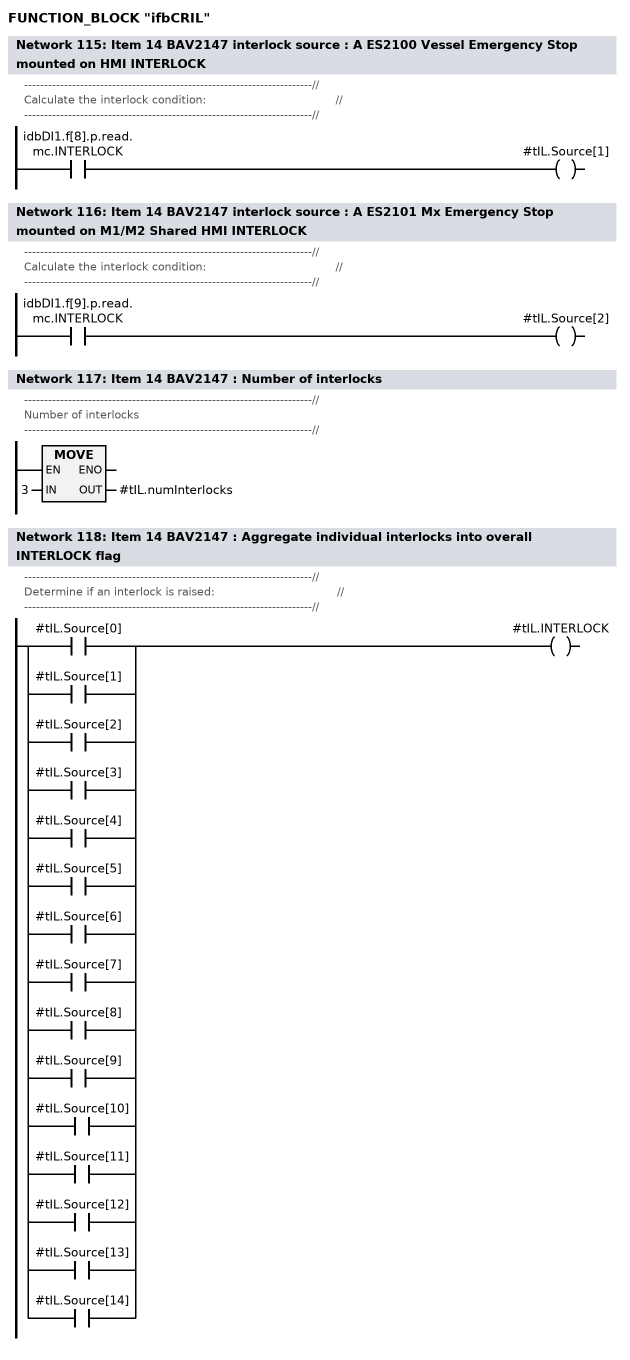
    A idbDI1.f[8].p.read.mc.INTERLOCK;
    = #tIL.Source[1];

NETWORK
TITLE = Item 14 BAV2147 interlock source : A ES2101 Mx Emergency Stop mounted on M1/M2 Shared HMI INTERLOCK
    //------------------------------------------------------------------------//
    // Calculate the interlock condition:                                     //
    //------------------------------------------------------------------------//
    A idbDI1.f[9].p.read.mc.INTERLOCK;
    = #tIL.Source[2];


NETWORK
TITLE = Item 14 BAV2147 : Number of interlocks
    //------------------------------------------------------------------------//
    // Number of interlocks
    //------------------------------------------------------------------------//
    L 3;
    T #tIL.numInterlocks;

NETWORK
TITLE = Item 14 BAV2147 : Aggregate individual interlocks into overall INTERLOCK flag
    //------------------------------------------------------------------------//
    // Determine if an interlock is raised:                                   //
    //------------------------------------------------------------------------//
    O #tIL.Source[0];
    O #tIL.Source[1];
    O #tIL.Source[2];
    O #tIL.Source[3];
    O #tIL.Source[4];
    O #tIL.Source[5];
    O #tIL.Source[6];
    O #tIL.Source[7];
    O #tIL.Source[8];
    O #tIL.Source[9];
    O #tIL.Source[10];
    O #tIL.Source[11];
    O #tIL.Source[12];
    O #tIL.Source[13];
    O #tIL.Source[14];
    = #tIL.INTERLOCK;

NETWORK
TITLE = Item 14 BAV2147 : Update the instance data
    //------------------------------------------------------------------------//
    // Update the instance DB with the calculated interlock flags:            //
    //------------------------------------------------------------------------//
    CALL MOVE
    {value_type := 'Variant'}
    (   IN                   := #tIL ,
        OUT                  := #p[14]
    );

NETWORK
TITLE = Item 15 BAV2149 : SMFLx CIP Drain Valve initialise variables
    //------------------------------------------------------------------------//
    // CRITICAL INTERLOCK   CRITICAL INTERLOCK   CRITICAL INTERLOCK   CRITICA //
    // CRITICAL INTERLOCK   CRITICAL INTERLOCK   CRITICAL INTERLOCK   CRITICA //
    //                                                                        //
    // Clear the interlock flag:                                              //
    //------------------------------------------------------------------------//
    A "alwaysLow";
    = #tIL.INTERLOCK;

    //------------------------------------------------------------------------//
    // Clear all interlock values to initialise them to off:                  //
    //------------------------------------------------------------------------//
    CALL FILL_BLK
    {value_type := 'Bool', count_type := 'UInt'}
    (   IN                   := 0 ,
        COUNT                := 15 ,
        OUT                  := #tIL.Source[0]
    );


NETWORK
TITLE = Item 15 BAV2149 interlock source : A RD2101 Vessel Burst Disc ALARM
    //------------------------------------------------------------------------//
    // Calculate the interlock condition:                                     //
    //------------------------------------------------------------------------//
    A idbDI1.f[14].p.read.mc.INTERLOCK;
    = #tIL.Source[0];

NETWORK
TITLE = Item 15 BAV2149 interlock source : A ES2100 Vessel Emergency Stop mounted on HMI INTERLOCK
    //------------------------------------------------------------------------//
    // Calculate the interlock condition:                                     //
    //------------------------------------------------------------------------//
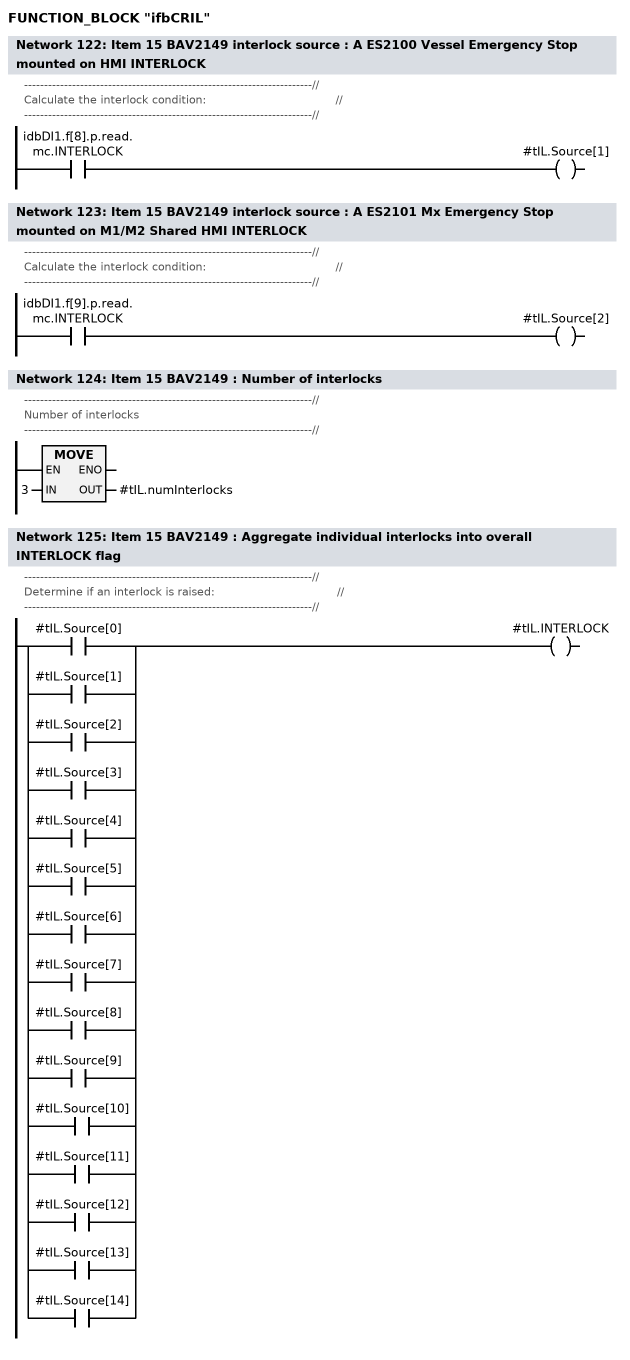
    A idbDI1.f[8].p.read.mc.INTERLOCK;
    = #tIL.Source[1];

NETWORK
TITLE = Item 15 BAV2149 interlock source : A ES2101 Mx Emergency Stop mounted on M1/M2 Shared HMI INTERLOCK
    //------------------------------------------------------------------------//
    // Calculate the interlock condition:                                     //
    //------------------------------------------------------------------------//
    A idbDI1.f[9].p.read.mc.INTERLOCK;
    = #tIL.Source[2];


NETWORK
TITLE = Item 15 BAV2149 : Number of interlocks
    //------------------------------------------------------------------------//
    // Number of interlocks
    //------------------------------------------------------------------------//
    L 3;
    T #tIL.numInterlocks;

NETWORK
TITLE = Item 15 BAV2149 : Aggregate individual interlocks into overall INTERLOCK flag
    //------------------------------------------------------------------------//
    // Determine if an interlock is raised:                                   //
    //------------------------------------------------------------------------//
    O #tIL.Source[0];
    O #tIL.Source[1];
    O #tIL.Source[2];
    O #tIL.Source[3];
    O #tIL.Source[4];
    O #tIL.Source[5];
    O #tIL.Source[6];
    O #tIL.Source[7];
    O #tIL.Source[8];
    O #tIL.Source[9];
    O #tIL.Source[10];
    O #tIL.Source[11];
    O #tIL.Source[12];
    O #tIL.Source[13];
    O #tIL.Source[14];
    = #tIL.INTERLOCK;

NETWORK
TITLE = Item 15 BAV2149 : Update the instance data
    //------------------------------------------------------------------------//
    // Update the instance DB with the calculated interlock flags:            //
    //------------------------------------------------------------------------//
    CALL MOVE
    {value_type := 'Variant'}
    (   IN                   := #tIL ,
        OUT                  := #p[15]
    );

NETWORK
TITLE = Item 16 BAV2167 : MMFLx Cooling Water Supply Drain Valve initialise variables
    //------------------------------------------------------------------------//
    // CRITICAL INTERLOCK   CRITICAL INTERLOCK   CRITICAL INTERLOCK   CRITICA //
    // CRITICAL INTERLOCK   CRITICAL INTERLOCK   CRITICAL INTERLOCK   CRITICA //
    //                                                                        //
    // Clear the interlock flag:                                              //
    //------------------------------------------------------------------------//
    A "alwaysLow";
    = #tIL.INTERLOCK;

    //------------------------------------------------------------------------//
    // Clear all interlock values to initialise them to off:                  //
    //------------------------------------------------------------------------//
    CALL FILL_BLK
    {value_type := 'Bool', count_type := 'UInt'}
    (   IN                   := 0 ,
        COUNT                := 15 ,
        OUT                  := #tIL.Source[0]
    );


NETWORK
TITLE = Item 16 BAV2167 interlock source : A RD2101 Vessel Burst Disc ALARM
    //------------------------------------------------------------------------//
    // Calculate the interlock condition:                                     //
    //------------------------------------------------------------------------//
    A idbDI1.f[14].p.read.mc.INTERLOCK;
    = #tIL.Source[0];

NETWORK
TITLE = Item 16 BAV2167 interlock source : A ES2100 Vessel Emergency Stop mounted on HMI INTERLOCK
    //------------------------------------------------------------------------//
    // Calculate the interlock condition:                                     //
    //------------------------------------------------------------------------//
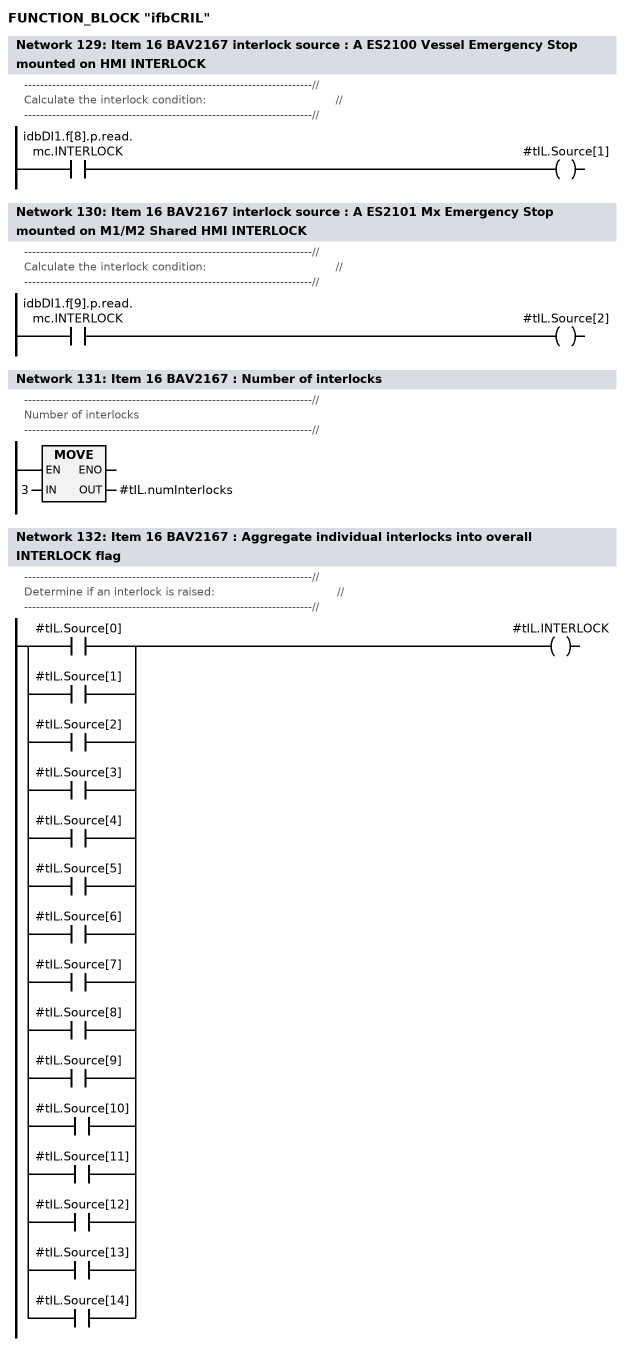
    A idbDI1.f[8].p.read.mc.INTERLOCK;
    = #tIL.Source[1];

NETWORK
TITLE = Item 16 BAV2167 interlock source : A ES2101 Mx Emergency Stop mounted on M1/M2 Shared HMI INTERLOCK
    //------------------------------------------------------------------------//
    // Calculate the interlock condition:                                     //
    //------------------------------------------------------------------------//
    A idbDI1.f[9].p.read.mc.INTERLOCK;
    = #tIL.Source[2];


NETWORK
TITLE = Item 16 BAV2167 : Number of interlocks
    //------------------------------------------------------------------------//
    // Number of interlocks
    //------------------------------------------------------------------------//
    L 3;
    T #tIL.numInterlocks;

NETWORK
TITLE = Item 16 BAV2167 : Aggregate individual interlocks into overall INTERLOCK flag
    //------------------------------------------------------------------------//
    // Determine if an interlock is raised:                                   //
    //------------------------------------------------------------------------//
    O #tIL.Source[0];
    O #tIL.Source[1];
    O #tIL.Source[2];
    O #tIL.Source[3];
    O #tIL.Source[4];
    O #tIL.Source[5];
    O #tIL.Source[6];
    O #tIL.Source[7];
    O #tIL.Source[8];
    O #tIL.Source[9];
    O #tIL.Source[10];
    O #tIL.Source[11];
    O #tIL.Source[12];
    O #tIL.Source[13];
    O #tIL.Source[14];
    = #tIL.INTERLOCK;

NETWORK
TITLE = Item 16 BAV2167 : Update the instance data
    //------------------------------------------------------------------------//
    // Update the instance DB with the calculated interlock flags:            //
    //------------------------------------------------------------------------//
    CALL MOVE
    {value_type := 'Variant'}
    (   IN                   := #tIL ,
        OUT                  := #p[16]
    );

NETWORK
TITLE = Item 17 BAV2169 : MMFLx Cooling Water Return Drain Valve initialise variables
    //------------------------------------------------------------------------//
    // CRITICAL INTERLOCK   CRITICAL INTERLOCK   CRITICAL INTERLOCK   CRITICA //
    // CRITICAL INTERLOCK   CRITICAL INTERLOCK   CRITICAL INTERLOCK   CRITICA //
    //                                                                        //
    // Clear the interlock flag:                                              //
    //------------------------------------------------------------------------//
    A "alwaysLow";
    = #tIL.INTERLOCK;

    //------------------------------------------------------------------------//
    // Clear all interlock values to initialise them to off:                  //
    //------------------------------------------------------------------------//
    CALL FILL_BLK
    {value_type := 'Bool', count_type := 'UInt'}
    (   IN                   := 0 ,
        COUNT                := 15 ,
        OUT                  := #tIL.Source[0]
    );


NETWORK
TITLE = Item 17 BAV2169 interlock source : A RD2101 Vessel Burst Disc ALARM
    //------------------------------------------------------------------------//
    // Calculate the interlock condition:                                     //
    //------------------------------------------------------------------------//
    A idbDI1.f[14].p.read.mc.INTERLOCK;
    = #tIL.Source[0];

NETWORK
TITLE = Item 17 BAV2169 interlock source : A ES2100 Vessel Emergency Stop mounted on HMI INTERLOCK
    //------------------------------------------------------------------------//
    // Calculate the interlock condition:                                     //
    //------------------------------------------------------------------------//
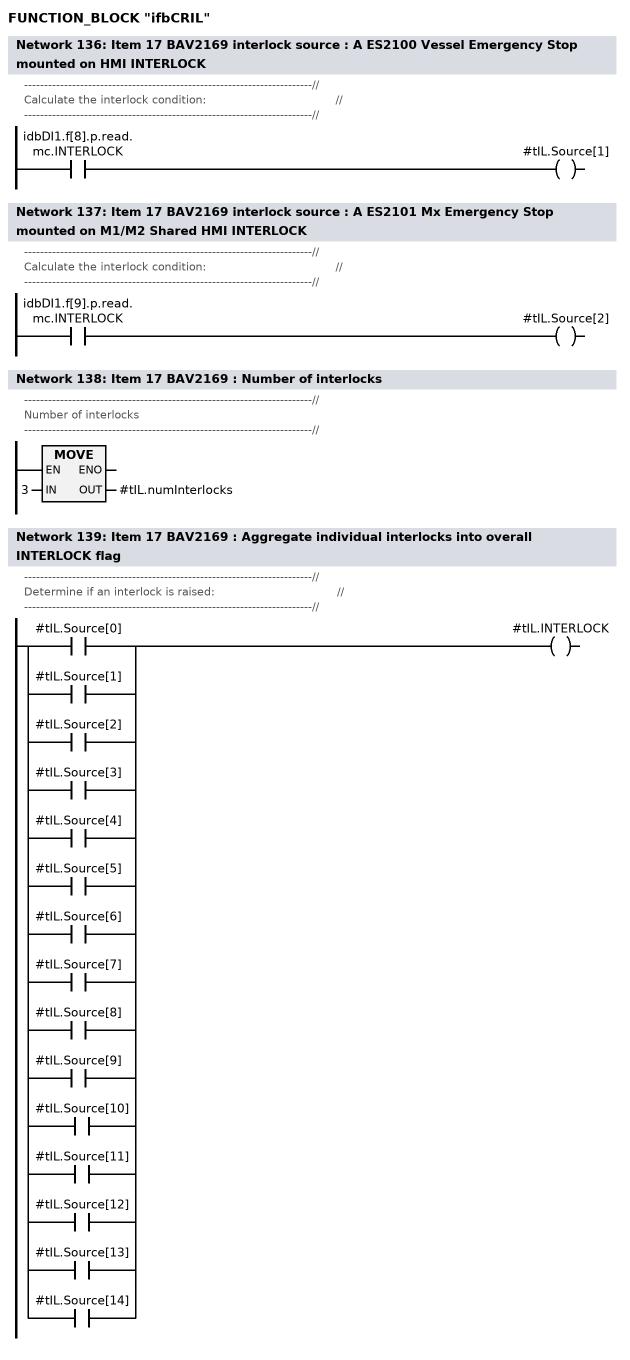
    A idbDI1.f[8].p.read.mc.INTERLOCK;
    = #tIL.Source[1];

NETWORK
TITLE = Item 17 BAV2169 interlock source : A ES2101 Mx Emergency Stop mounted on M1/M2 Shared HMI INTERLOCK
    //------------------------------------------------------------------------//
    // Calculate the interlock condition:                                     //
    //------------------------------------------------------------------------//
    A idbDI1.f[9].p.read.mc.INTERLOCK;
    = #tIL.Source[2];


NETWORK
TITLE = Item 17 BAV2169 : Number of interlocks
    //------------------------------------------------------------------------//
    // Number of interlocks
    //------------------------------------------------------------------------//
    L 3;
    T #tIL.numInterlocks;

NETWORK
TITLE = Item 17 BAV2169 : Aggregate individual interlocks into overall INTERLOCK flag
    //------------------------------------------------------------------------//
    // Determine if an interlock is raised:                                   //
    //------------------------------------------------------------------------//
    O #tIL.Source[0];
    O #tIL.Source[1];
    O #tIL.Source[2];
    O #tIL.Source[3];
    O #tIL.Source[4];
    O #tIL.Source[5];
    O #tIL.Source[6];
    O #tIL.Source[7];
    O #tIL.Source[8];
    O #tIL.Source[9];
    O #tIL.Source[10];
    O #tIL.Source[11];
    O #tIL.Source[12];
    O #tIL.Source[13];
    O #tIL.Source[14];
    = #tIL.INTERLOCK;

NETWORK
TITLE = Item 17 BAV2169 : Update the instance data
    //------------------------------------------------------------------------//
    // Update the instance DB with the calculated interlock flags:            //
    //------------------------------------------------------------------------//
    CALL MOVE
    {value_type := 'Variant'}
    (   IN                   := #tIL ,
        OUT                  := #p[17]
    );

NETWORK
TITLE = Item 18 BAV3139 : Vent line drain valve initialise variables
    //------------------------------------------------------------------------//
    // CRITICAL INTERLOCK   CRITICAL INTERLOCK   CRITICAL INTERLOCK   CRITICA //
    // CRITICAL INTERLOCK   CRITICAL INTERLOCK   CRITICAL INTERLOCK   CRITICA //
    //                                                                        //
    // Clear the interlock flag:                                              //
    //------------------------------------------------------------------------//
    A "alwaysLow";
    = #tIL.INTERLOCK;

    //------------------------------------------------------------------------//
    // Clear all interlock values to initialise them to off:                  //
    //------------------------------------------------------------------------//
    CALL FILL_BLK
    {value_type := 'Bool', count_type := 'UInt'}
    (   IN                   := 0 ,
        COUNT                := 15 ,
        OUT                  := #tIL.Source[0]
    );


NETWORK
TITLE = Item 18 BAV3139 interlock source : A RD3101 Vessel Burst Disc ALARM
    //------------------------------------------------------------------------//
    // Calculate the interlock condition:                                     //
    //------------------------------------------------------------------------//
    A idbDI1.f[15].p.read.mc.INTERLOCK;
    = #tIL.Source[0];

NETWORK
TITLE = Item 18 BAV3139 interlock source : A ES3100 Vessel Emergency Stop mounted on HMI INTERLOCK
    //------------------------------------------------------------------------//
    // Calculate the interlock condition:                                     //
    //------------------------------------------------------------------------//
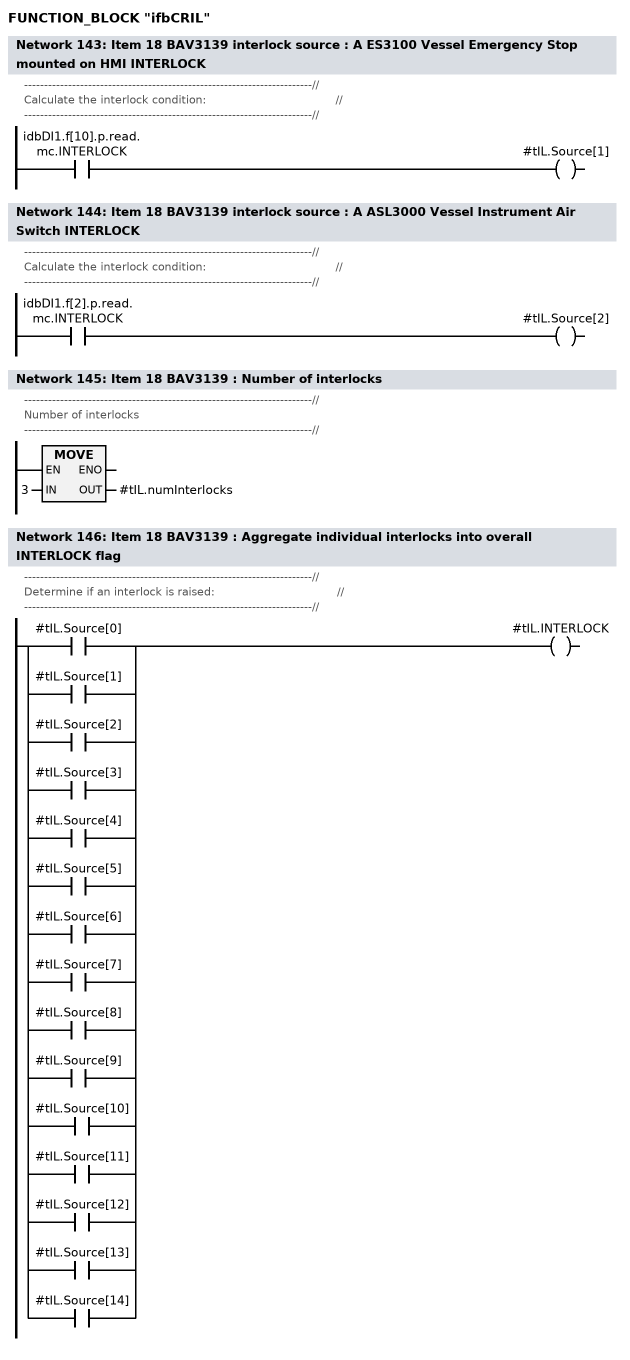
    A idbDI1.f[10].p.read.mc.INTERLOCK;
    = #tIL.Source[1];

NETWORK
TITLE = Item 18 BAV3139 interlock source : A ASL3000 Vessel Instrument Air Switch INTERLOCK
    //------------------------------------------------------------------------//
    // Calculate the interlock condition:                                     //
    //------------------------------------------------------------------------//
    A idbDI1.f[2].p.read.mc.INTERLOCK;
    = #tIL.Source[2];


NETWORK
TITLE = Item 18 BAV3139 : Number of interlocks
    //------------------------------------------------------------------------//
    // Number of interlocks
    //------------------------------------------------------------------------//
    L 3;
    T #tIL.numInterlocks;

NETWORK
TITLE = Item 18 BAV3139 : Aggregate individual interlocks into overall INTERLOCK flag
    //------------------------------------------------------------------------//
    // Determine if an interlock is raised:                                   //
    //------------------------------------------------------------------------//
    O #tIL.Source[0];
    O #tIL.Source[1];
    O #tIL.Source[2];
    O #tIL.Source[3];
    O #tIL.Source[4];
    O #tIL.Source[5];
    O #tIL.Source[6];
    O #tIL.Source[7];
    O #tIL.Source[8];
    O #tIL.Source[9];
    O #tIL.Source[10];
    O #tIL.Source[11];
    O #tIL.Source[12];
    O #tIL.Source[13];
    O #tIL.Source[14];
    = #tIL.INTERLOCK;

NETWORK
TITLE = Item 18 BAV3139 : Update the instance data
    //------------------------------------------------------------------------//
    // Update the instance DB with the calculated interlock flags:            //
    //------------------------------------------------------------------------//
    CALL MOVE
    {value_type := 'Variant'}
    (   IN                   := #tIL ,
        OUT                  := #p[18]
    );

NETWORK
TITLE = Item 19 BAV3141 : Vent Filter Drain valve initialise variables
    //------------------------------------------------------------------------//
    // CRITICAL INTERLOCK   CRITICAL INTERLOCK   CRITICAL INTERLOCK   CRITICA //
    // CRITICAL INTERLOCK   CRITICAL INTERLOCK   CRITICAL INTERLOCK   CRITICA //
    //                                                                        //
    // Clear the interlock flag:                                              //
    //------------------------------------------------------------------------//
    A "alwaysLow";
    = #tIL.INTERLOCK;

    //------------------------------------------------------------------------//
    // Clear all interlock values to initialise them to off:                  //
    //------------------------------------------------------------------------//
    CALL FILL_BLK
    {value_type := 'Bool', count_type := 'UInt'}
    (   IN                   := 0 ,
        COUNT                := 15 ,
        OUT                  := #tIL.Source[0]
    );


NETWORK
TITLE = Item 19 BAV3141 interlock source : A RD3101 Vessel Burst Disc ALARM
    //------------------------------------------------------------------------//
    // Calculate the interlock condition:                                     //
    //------------------------------------------------------------------------//
    A idbDI1.f[15].p.read.mc.INTERLOCK;
    = #tIL.Source[0];

NETWORK
TITLE = Item 19 BAV3141 interlock source : A ES3100 Vessel Emergency Stop mounted on HMI INTERLOCK
    //------------------------------------------------------------------------//
    // Calculate the interlock condition:                                     //
    //------------------------------------------------------------------------//
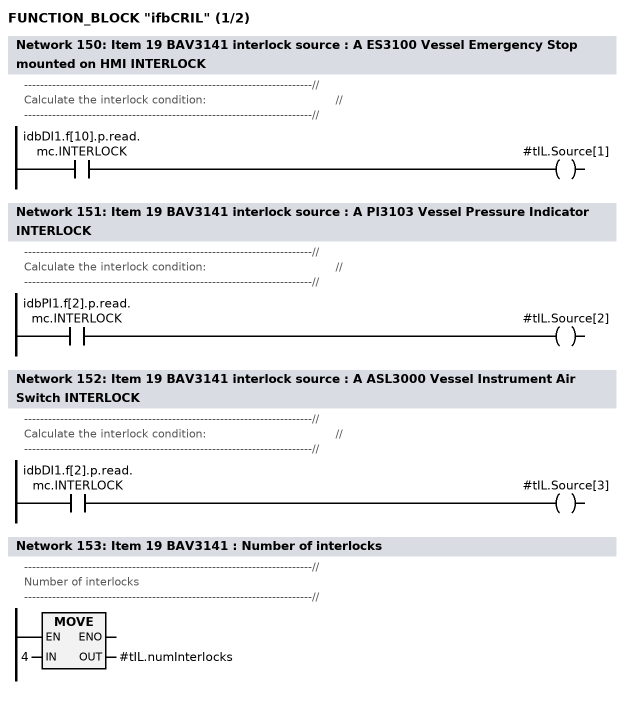
    A idbDI1.f[10].p.read.mc.INTERLOCK;
    = #tIL.Source[1];

NETWORK
TITLE = Item 19 BAV3141 interlock source : A PI3103 Vessel Pressure Indicator INTERLOCK
    //------------------------------------------------------------------------//
    // Calculate the interlock condition:                                     //
    //------------------------------------------------------------------------//
    A idbPI1.f[2].p.read.mc.INTERLOCK;
    = #tIL.Source[2];

NETWORK
TITLE = Item 19 BAV3141 interlock source : A ASL3000 Vessel Instrument Air Switch INTERLOCK
    //------------------------------------------------------------------------//
    // Calculate the interlock condition:                                     //
    //------------------------------------------------------------------------//
    A idbDI1.f[2].p.read.mc.INTERLOCK;
    = #tIL.Source[3];


NETWORK
TITLE = Item 19 BAV3141 : Number of interlocks
    //------------------------------------------------------------------------//
    // Number of interlocks
    //------------------------------------------------------------------------//
    L 4;
    T #tIL.numInterlocks;

NETWORK
TITLE = Item 19 BAV3141 : Aggregate individual interlocks into overall INTERLOCK flag
    //------------------------------------------------------------------------//
    // Determine if an interlock is raised:                                   //
    //------------------------------------------------------------------------//
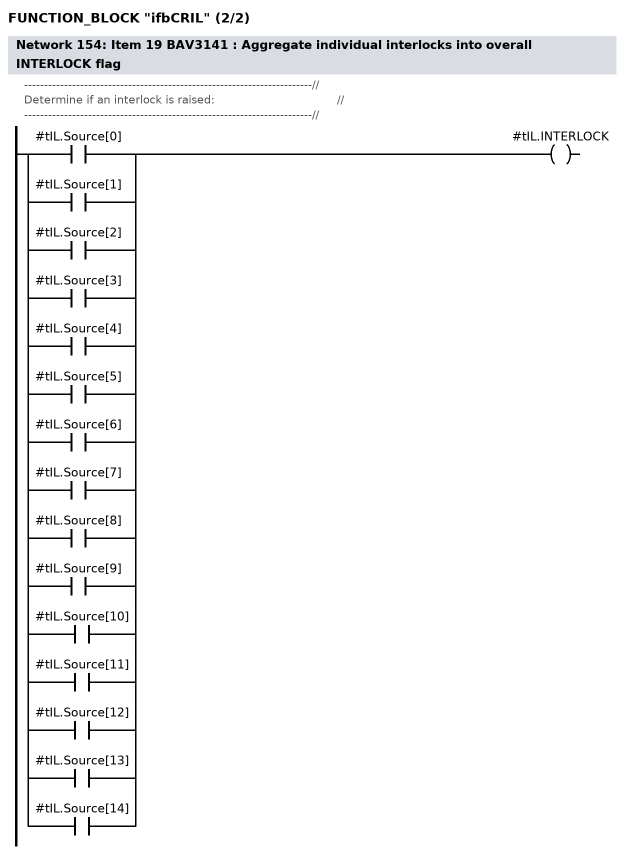
    O #tIL.Source[0];
    O #tIL.Source[1];
    O #tIL.Source[2];
    O #tIL.Source[3];
    O #tIL.Source[4];
    O #tIL.Source[5];
    O #tIL.Source[6];
    O #tIL.Source[7];
    O #tIL.Source[8];
    O #tIL.Source[9];
    O #tIL.Source[10];
    O #tIL.Source[11];
    O #tIL.Source[12];
    O #tIL.Source[13];
    O #tIL.Source[14];
    = #tIL.INTERLOCK;

NETWORK
TITLE = Item 19 BAV3141 : Update the instance data
    //------------------------------------------------------------------------//
    // Update the instance DB with the calculated interlock flags:            //
    //------------------------------------------------------------------------//
    CALL MOVE
    {value_type := 'Variant'}
    (   IN                   := #tIL ,
        OUT                  := #p[19]
    );

NETWORK
TITLE = Item 20 BAV3143 : SIP Condensate Drain Valve initialise variables
    //------------------------------------------------------------------------//
    // CRITICAL INTERLOCK   CRITICAL INTERLOCK   CRITICAL INTERLOCK   CRITICA //
    // CRITICAL INTERLOCK   CRITICAL INTERLOCK   CRITICAL INTERLOCK   CRITICA //
    //                                                                        //
    // Clear the interlock flag:                                              //
    //------------------------------------------------------------------------//
    A "alwaysLow";
    = #tIL.INTERLOCK;

    //------------------------------------------------------------------------//
    // Clear all interlock values to initialise them to off:                  //
    //------------------------------------------------------------------------//
    CALL FILL_BLK
    {value_type := 'Bool', count_type := 'UInt'}
    (   IN                   := 0 ,
        COUNT                := 15 ,
        OUT                  := #tIL.Source[0]
    );


NETWORK
TITLE = Item 20 BAV3143 interlock source : A RD3101 Vessel Burst Disc ALARM
    //------------------------------------------------------------------------//
    // Calculate the interlock condition:                                     //
    //------------------------------------------------------------------------//
    A idbDI1.f[15].p.read.mc.INTERLOCK;
    = #tIL.Source[0];

NETWORK
TITLE = Item 20 BAV3143 interlock source : A ES3100 Vessel Emergency Stop mounted on HMI INTERLOCK
    //------------------------------------------------------------------------//
    // Calculate the interlock condition:                                     //
    //------------------------------------------------------------------------//
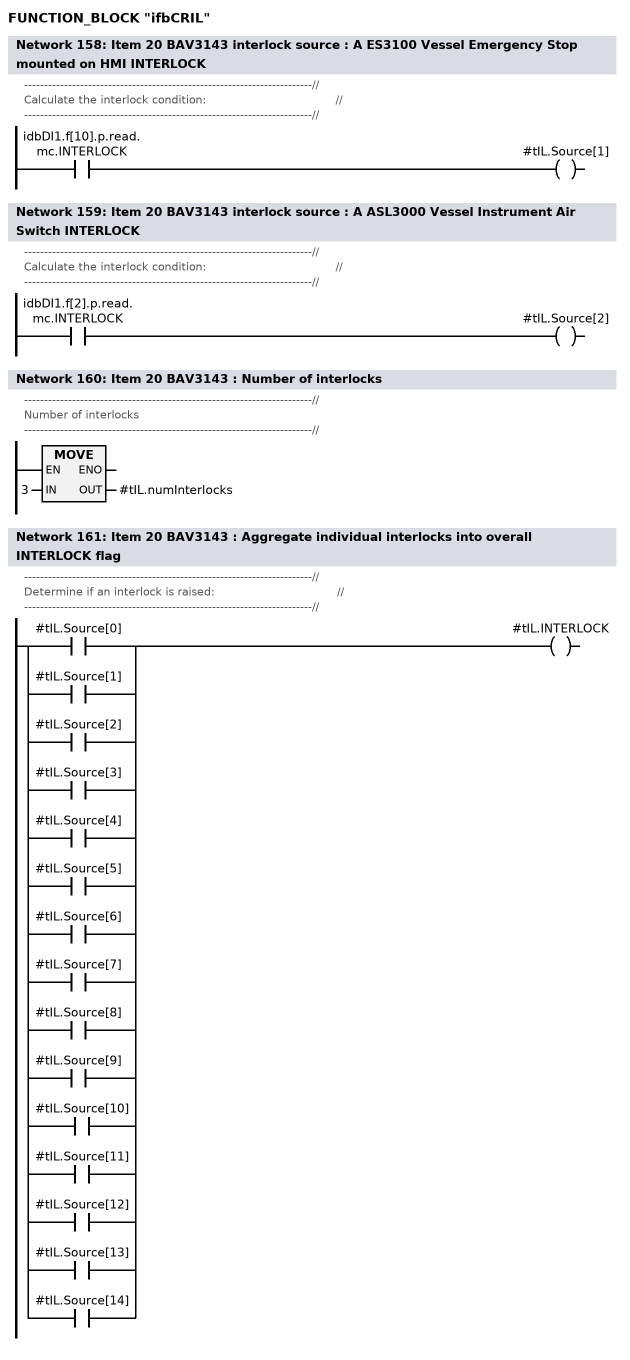
    A idbDI1.f[10].p.read.mc.INTERLOCK;
    = #tIL.Source[1];

NETWORK
TITLE = Item 20 BAV3143 interlock source : A ASL3000 Vessel Instrument Air Switch INTERLOCK
    //------------------------------------------------------------------------//
    // Calculate the interlock condition:                                     //
    //------------------------------------------------------------------------//
    A idbDI1.f[2].p.read.mc.INTERLOCK;
    = #tIL.Source[2];


NETWORK
TITLE = Item 20 BAV3143 : Number of interlocks
    //------------------------------------------------------------------------//
    // Number of interlocks
    //------------------------------------------------------------------------//
    L 3;
    T #tIL.numInterlocks;

NETWORK
TITLE = Item 20 BAV3143 : Aggregate individual interlocks into overall INTERLOCK flag
    //------------------------------------------------------------------------//
    // Determine if an interlock is raised:                                   //
    //------------------------------------------------------------------------//
    O #tIL.Source[0];
    O #tIL.Source[1];
    O #tIL.Source[2];
    O #tIL.Source[3];
    O #tIL.Source[4];
    O #tIL.Source[5];
    O #tIL.Source[6];
    O #tIL.Source[7];
    O #tIL.Source[8];
    O #tIL.Source[9];
    O #tIL.Source[10];
    O #tIL.Source[11];
    O #tIL.Source[12];
    O #tIL.Source[13];
    O #tIL.Source[14];
    = #tIL.INTERLOCK;

NETWORK
TITLE = Item 20 BAV3143 : Update the instance data
    //------------------------------------------------------------------------//
    // Update the instance DB with the calculated interlock flags:            //
    //------------------------------------------------------------------------//
    CALL MOVE
    {value_type := 'Variant'}
    (   IN                   := #tIL ,
        OUT                  := #p[20]
    );

NETWORK
TITLE = Item 21 BAV3145 : CIP Drain Valve initialise variables
    //------------------------------------------------------------------------//
    // CRITICAL INTERLOCK   CRITICAL INTERLOCK   CRITICAL INTERLOCK   CRITICA //
    // CRITICAL INTERLOCK   CRITICAL INTERLOCK   CRITICAL INTERLOCK   CRITICA //
    //                                                                        //
    // Clear the interlock flag:                                              //
    //------------------------------------------------------------------------//
    A "alwaysLow";
    = #tIL.INTERLOCK;

    //------------------------------------------------------------------------//
    // Clear all interlock values to initialise them to off:                  //
    //------------------------------------------------------------------------//
    CALL FILL_BLK
    {value_type := 'Bool', count_type := 'UInt'}
    (   IN                   := 0 ,
        COUNT                := 15 ,
        OUT                  := #tIL.Source[0]
    );


NETWORK
TITLE = Item 21 BAV3145 interlock source : A RD3101 Vessel Burst Disc ALARM
    //------------------------------------------------------------------------//
    // Calculate the interlock condition:                                     //
    //------------------------------------------------------------------------//
    A idbDI1.f[15].p.read.mc.INTERLOCK;
    = #tIL.Source[0];

NETWORK
TITLE = Item 21 BAV3145 interlock source : A ES3100 Vessel Emergency Stop mounted on HMI INTERLOCK
    //------------------------------------------------------------------------//
    // Calculate the interlock condition:                                     //
    //------------------------------------------------------------------------//
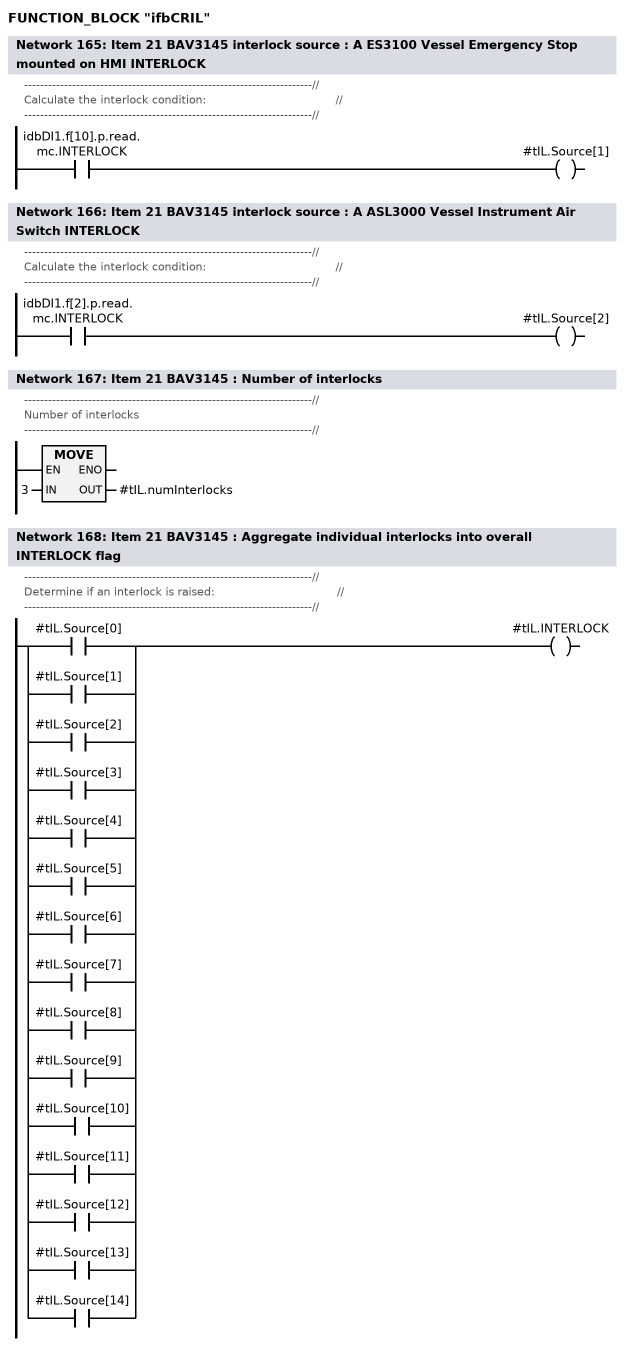
    A idbDI1.f[10].p.read.mc.INTERLOCK;
    = #tIL.Source[1];

NETWORK
TITLE = Item 21 BAV3145 interlock source : A ASL3000 Vessel Instrument Air Switch INTERLOCK
    //------------------------------------------------------------------------//
    // Calculate the interlock condition:                                     //
    //------------------------------------------------------------------------//
    A idbDI1.f[2].p.read.mc.INTERLOCK;
    = #tIL.Source[2];


NETWORK
TITLE = Item 21 BAV3145 : Number of interlocks
    //------------------------------------------------------------------------//
    // Number of interlocks
    //------------------------------------------------------------------------//
    L 3;
    T #tIL.numInterlocks;

NETWORK
TITLE = Item 21 BAV3145 : Aggregate individual interlocks into overall INTERLOCK flag
    //------------------------------------------------------------------------//
    // Determine if an interlock is raised:                                   //
    //------------------------------------------------------------------------//
    O #tIL.Source[0];
    O #tIL.Source[1];
    O #tIL.Source[2];
    O #tIL.Source[3];
    O #tIL.Source[4];
    O #tIL.Source[5];
    O #tIL.Source[6];
    O #tIL.Source[7];
    O #tIL.Source[8];
    O #tIL.Source[9];
    O #tIL.Source[10];
    O #tIL.Source[11];
    O #tIL.Source[12];
    O #tIL.Source[13];
    O #tIL.Source[14];
    = #tIL.INTERLOCK;

NETWORK
TITLE = Item 21 BAV3145 : Update the instance data
    //------------------------------------------------------------------------//
    // Update the instance DB with the calculated interlock flags:            //
    //------------------------------------------------------------------------//
    CALL MOVE
    {value_type := 'Variant'}
    (   IN                   := #tIL ,
        OUT                  := #p[21]
    );

NETWORK
TITLE = Item 22 BAV4139 : Vent line drain valve initialise variables
    //------------------------------------------------------------------------//
    // CRITICAL INTERLOCK   CRITICAL INTERLOCK   CRITICAL INTERLOCK   CRITICA //
    // CRITICAL INTERLOCK   CRITICAL INTERLOCK   CRITICAL INTERLOCK   CRITICA //
    //                                                                        //
    // Clear the interlock flag:                                              //
    //------------------------------------------------------------------------//
    A "alwaysLow";
    = #tIL.INTERLOCK;

    //------------------------------------------------------------------------//
    // Clear all interlock values to initialise them to off:                  //
    //------------------------------------------------------------------------//
    CALL FILL_BLK
    {value_type := 'Bool', count_type := 'UInt'}
    (   IN                   := 0 ,
        COUNT                := 15 ,
        OUT                  := #tIL.Source[0]
    );


NETWORK
TITLE = Item 22 BAV4139 interlock source : A RD4101 Vessel Burst Disc ALARM
    //------------------------------------------------------------------------//
    // Calculate the interlock condition:                                     //
    //------------------------------------------------------------------------//
    A idbDI1.f[16].p.read.mc.INTERLOCK;
    = #tIL.Source[0];

NETWORK
TITLE = Item 22 BAV4139 interlock source : A ES4100 Vessel Emergency Stop mounted on HMI INTERLOCK
    //------------------------------------------------------------------------//
    // Calculate the interlock condition:                                     //
    //------------------------------------------------------------------------//
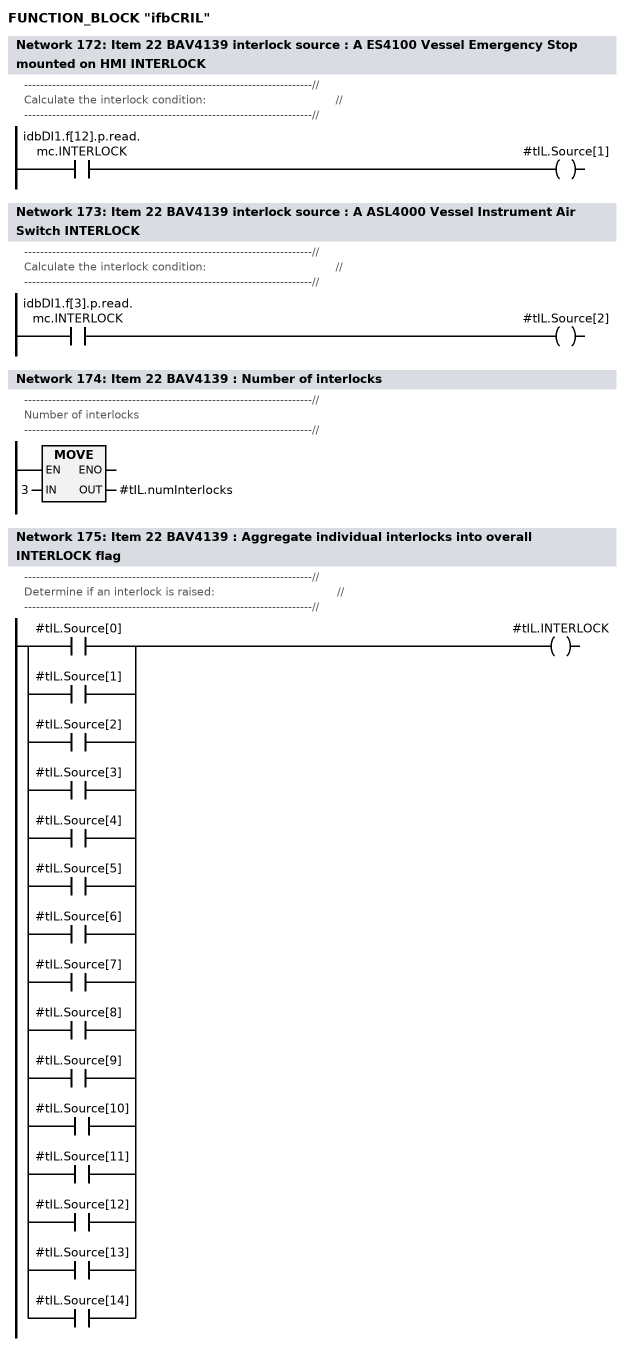
    A idbDI1.f[12].p.read.mc.INTERLOCK;
    = #tIL.Source[1];

NETWORK
TITLE = Item 22 BAV4139 interlock source : A ASL4000 Vessel Instrument Air Switch INTERLOCK
    //------------------------------------------------------------------------//
    // Calculate the interlock condition:                                     //
    //------------------------------------------------------------------------//
    A idbDI1.f[3].p.read.mc.INTERLOCK;
    = #tIL.Source[2];


NETWORK
TITLE = Item 22 BAV4139 : Number of interlocks
    //------------------------------------------------------------------------//
    // Number of interlocks
    //------------------------------------------------------------------------//
    L 3;
    T #tIL.numInterlocks;

NETWORK
TITLE = Item 22 BAV4139 : Aggregate individual interlocks into overall INTERLOCK flag
    //------------------------------------------------------------------------//
    // Determine if an interlock is raised:                                   //
    //------------------------------------------------------------------------//
    O #tIL.Source[0];
    O #tIL.Source[1];
    O #tIL.Source[2];
    O #tIL.Source[3];
    O #tIL.Source[4];
    O #tIL.Source[5];
    O #tIL.Source[6];
    O #tIL.Source[7];
    O #tIL.Source[8];
    O #tIL.Source[9];
    O #tIL.Source[10];
    O #tIL.Source[11];
    O #tIL.Source[12];
    O #tIL.Source[13];
    O #tIL.Source[14];
    = #tIL.INTERLOCK;

NETWORK
TITLE = Item 22 BAV4139 : Update the instance data
    //------------------------------------------------------------------------//
    // Update the instance DB with the calculated interlock flags:            //
    //------------------------------------------------------------------------//
    CALL MOVE
    {value_type := 'Variant'}
    (   IN                   := #tIL ,
        OUT                  := #p[22]
    );

NETWORK
TITLE = Item 23 BAV4141 : Vent Filter Drain valve initialise variables
    //------------------------------------------------------------------------//
    // CRITICAL INTERLOCK   CRITICAL INTERLOCK   CRITICAL INTERLOCK   CRITICA //
    // CRITICAL INTERLOCK   CRITICAL INTERLOCK   CRITICAL INTERLOCK   CRITICA //
    //                                                                        //
    // Clear the interlock flag:                                              //
    //------------------------------------------------------------------------//
    A "alwaysLow";
    = #tIL.INTERLOCK;

    //------------------------------------------------------------------------//
    // Clear all interlock values to initialise them to off:                  //
    //------------------------------------------------------------------------//
    CALL FILL_BLK
    {value_type := 'Bool', count_type := 'UInt'}
    (   IN                   := 0 ,
        COUNT                := 15 ,
        OUT                  := #tIL.Source[0]
    );


NETWORK
TITLE = Item 23 BAV4141 interlock source : A RD4101 Vessel Burst Disc ALARM
    //------------------------------------------------------------------------//
    // Calculate the interlock condition:                                     //
    //------------------------------------------------------------------------//
    A idbDI1.f[16].p.read.mc.INTERLOCK;
    = #tIL.Source[0];

NETWORK
TITLE = Item 23 BAV4141 interlock source : A ES4100 Vessel Emergency Stop mounted on HMI INTERLOCK
    //------------------------------------------------------------------------//
    // Calculate the interlock condition:                                     //
    //------------------------------------------------------------------------//
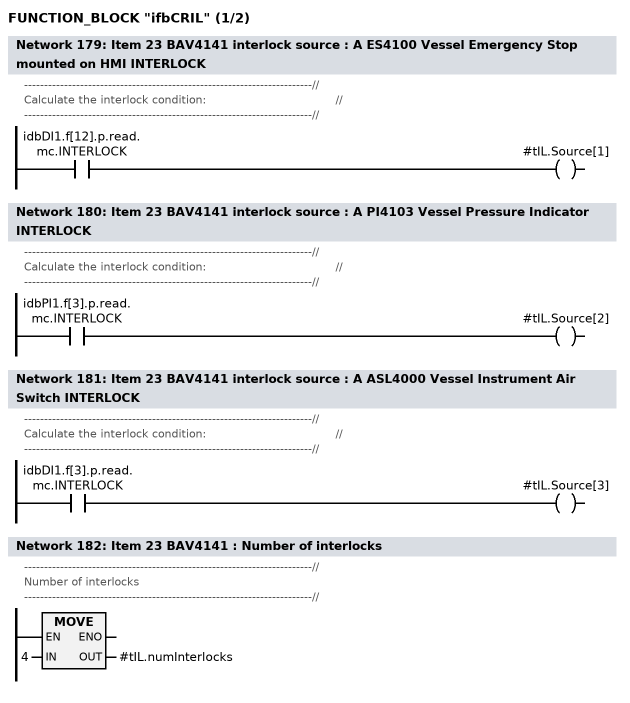
    A idbDI1.f[12].p.read.mc.INTERLOCK;
    = #tIL.Source[1];

NETWORK
TITLE = Item 23 BAV4141 interlock source : A PI4103 Vessel Pressure Indicator INTERLOCK
    //------------------------------------------------------------------------//
    // Calculate the interlock condition:                                     //
    //------------------------------------------------------------------------//
    A idbPI1.f[3].p.read.mc.INTERLOCK;
    = #tIL.Source[2];

NETWORK
TITLE = Item 23 BAV4141 interlock source : A ASL4000 Vessel Instrument Air Switch INTERLOCK
    //------------------------------------------------------------------------//
    // Calculate the interlock condition:                                     //
    //------------------------------------------------------------------------//
    A idbDI1.f[3].p.read.mc.INTERLOCK;
    = #tIL.Source[3];


NETWORK
TITLE = Item 23 BAV4141 : Number of interlocks
    //------------------------------------------------------------------------//
    // Number of interlocks
    //------------------------------------------------------------------------//
    L 4;
    T #tIL.numInterlocks;

NETWORK
TITLE = Item 23 BAV4141 : Aggregate individual interlocks into overall INTERLOCK flag
    //------------------------------------------------------------------------//
    // Determine if an interlock is raised:                                   //
    //------------------------------------------------------------------------//
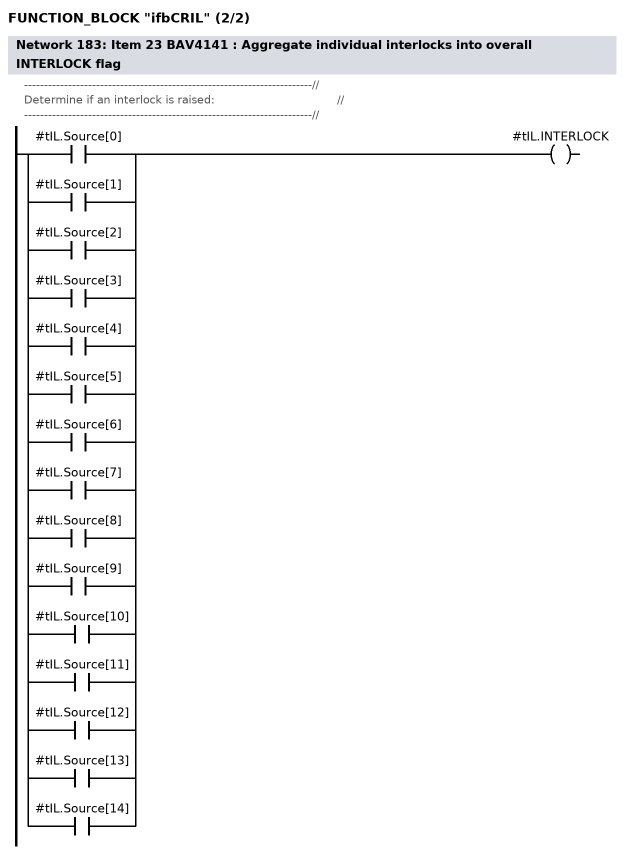
    O #tIL.Source[0];
    O #tIL.Source[1];
    O #tIL.Source[2];
    O #tIL.Source[3];
    O #tIL.Source[4];
    O #tIL.Source[5];
    O #tIL.Source[6];
    O #tIL.Source[7];
    O #tIL.Source[8];
    O #tIL.Source[9];
    O #tIL.Source[10];
    O #tIL.Source[11];
    O #tIL.Source[12];
    O #tIL.Source[13];
    O #tIL.Source[14];
    = #tIL.INTERLOCK;

NETWORK
TITLE = Item 23 BAV4141 : Update the instance data
    //------------------------------------------------------------------------//
    // Update the instance DB with the calculated interlock flags:            //
    //------------------------------------------------------------------------//
    CALL MOVE
    {value_type := 'Variant'}
    (   IN                   := #tIL ,
        OUT                  := #p[23]
    );

NETWORK
TITLE = Item 24 BAV4143 : SIP Condensate Drain Valve initialise variables
    //------------------------------------------------------------------------//
    // CRITICAL INTERLOCK   CRITICAL INTERLOCK   CRITICAL INTERLOCK   CRITICA //
    // CRITICAL INTERLOCK   CRITICAL INTERLOCK   CRITICAL INTERLOCK   CRITICA //
    //                                                                        //
    // Clear the interlock flag:                                              //
    //------------------------------------------------------------------------//
    A "alwaysLow";
    = #tIL.INTERLOCK;

    //------------------------------------------------------------------------//
    // Clear all interlock values to initialise them to off:                  //
    //------------------------------------------------------------------------//
    CALL FILL_BLK
    {value_type := 'Bool', count_type := 'UInt'}
    (   IN                   := 0 ,
        COUNT                := 15 ,
        OUT                  := #tIL.Source[0]
    );


NETWORK
TITLE = Item 24 BAV4143 interlock source : A RD4101 Vessel Burst Disc ALARM
    //------------------------------------------------------------------------//
    // Calculate the interlock condition:                                     //
    //------------------------------------------------------------------------//
    A idbDI1.f[16].p.read.mc.INTERLOCK;
    = #tIL.Source[0];

NETWORK
TITLE = Item 24 BAV4143 interlock source : A ES4100 Vessel Emergency Stop mounted on HMI INTERLOCK
    //------------------------------------------------------------------------//
    // Calculate the interlock condition:                                     //
    //------------------------------------------------------------------------//
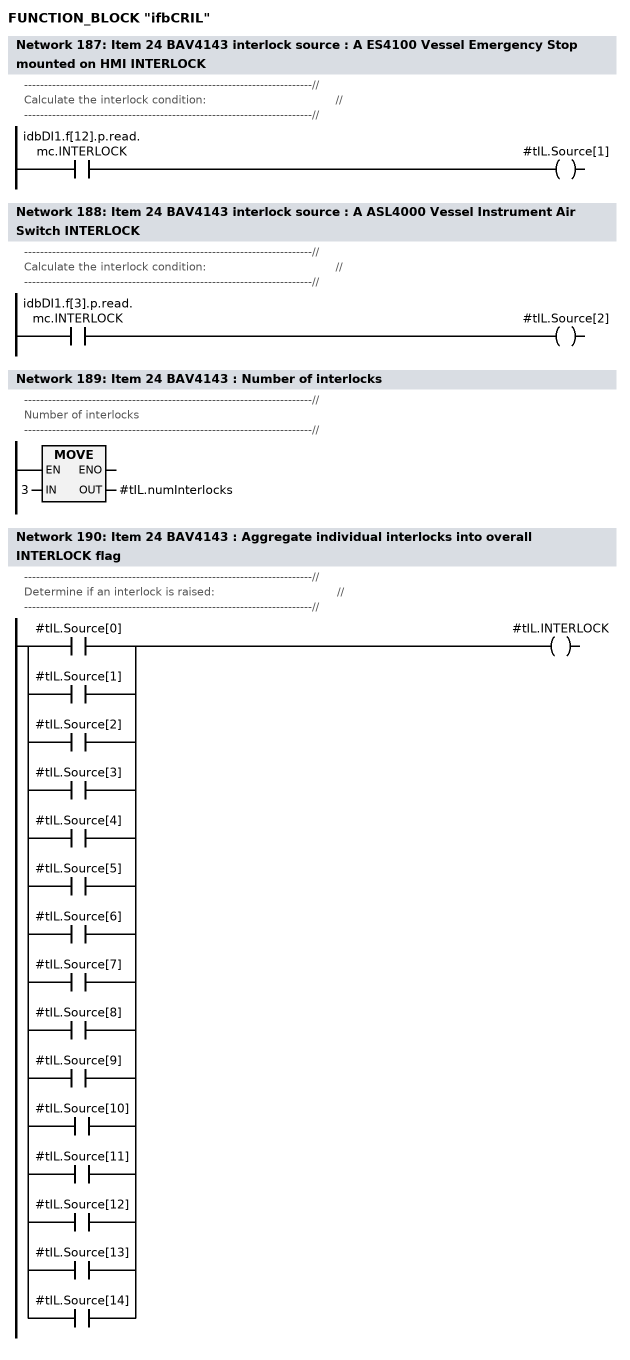
    A idbDI1.f[12].p.read.mc.INTERLOCK;
    = #tIL.Source[1];

NETWORK
TITLE = Item 24 BAV4143 interlock source : A ASL4000 Vessel Instrument Air Switch INTERLOCK
    //------------------------------------------------------------------------//
    // Calculate the interlock condition:                                     //
    //------------------------------------------------------------------------//
    A idbDI1.f[3].p.read.mc.INTERLOCK;
    = #tIL.Source[2];


NETWORK
TITLE = Item 24 BAV4143 : Number of interlocks
    //------------------------------------------------------------------------//
    // Number of interlocks
    //------------------------------------------------------------------------//
    L 3;
    T #tIL.numInterlocks;

NETWORK
TITLE = Item 24 BAV4143 : Aggregate individual interlocks into overall INTERLOCK flag
    //------------------------------------------------------------------------//
    // Determine if an interlock is raised:                                   //
    //------------------------------------------------------------------------//
    O #tIL.Source[0];
    O #tIL.Source[1];
    O #tIL.Source[2];
    O #tIL.Source[3];
    O #tIL.Source[4];
    O #tIL.Source[5];
    O #tIL.Source[6];
    O #tIL.Source[7];
    O #tIL.Source[8];
    O #tIL.Source[9];
    O #tIL.Source[10];
    O #tIL.Source[11];
    O #tIL.Source[12];
    O #tIL.Source[13];
    O #tIL.Source[14];
    = #tIL.INTERLOCK;

NETWORK
TITLE = Item 24 BAV4143 : Update the instance data
    //------------------------------------------------------------------------//
    // Update the instance DB with the calculated interlock flags:            //
    //------------------------------------------------------------------------//
    CALL MOVE
    {value_type := 'Variant'}
    (   IN                   := #tIL ,
        OUT                  := #p[24]
    );

NETWORK
TITLE = Item 25 BAV4145 : CIP Drain Valve initialise variables
    //------------------------------------------------------------------------//
    // CRITICAL INTERLOCK   CRITICAL INTERLOCK   CRITICAL INTERLOCK   CRITICA //
    // CRITICAL INTERLOCK   CRITICAL INTERLOCK   CRITICAL INTERLOCK   CRITICA //
    //                                                                        //
    // Clear the interlock flag:                                              //
    //------------------------------------------------------------------------//
    A "alwaysLow";
    = #tIL.INTERLOCK;

    //------------------------------------------------------------------------//
    // Clear all interlock values to initialise them to off:                  //
    //------------------------------------------------------------------------//
    CALL FILL_BLK
    {value_type := 'Bool', count_type := 'UInt'}
    (   IN                   := 0 ,
        COUNT                := 15 ,
        OUT                  := #tIL.Source[0]
    );


NETWORK
TITLE = Item 25 BAV4145 interlock source : A RD4101 Vessel Burst Disc ALARM
    //------------------------------------------------------------------------//
    // Calculate the interlock condition:                                     //
    //------------------------------------------------------------------------//
    A idbDI1.f[16].p.read.mc.INTERLOCK;
    = #tIL.Source[0];

NETWORK
TITLE = Item 25 BAV4145 interlock source : A ES4100 Vessel Emergency Stop mounted on HMI INTERLOCK
    //------------------------------------------------------------------------//
    // Calculate the interlock condition:                                     //
    //------------------------------------------------------------------------//
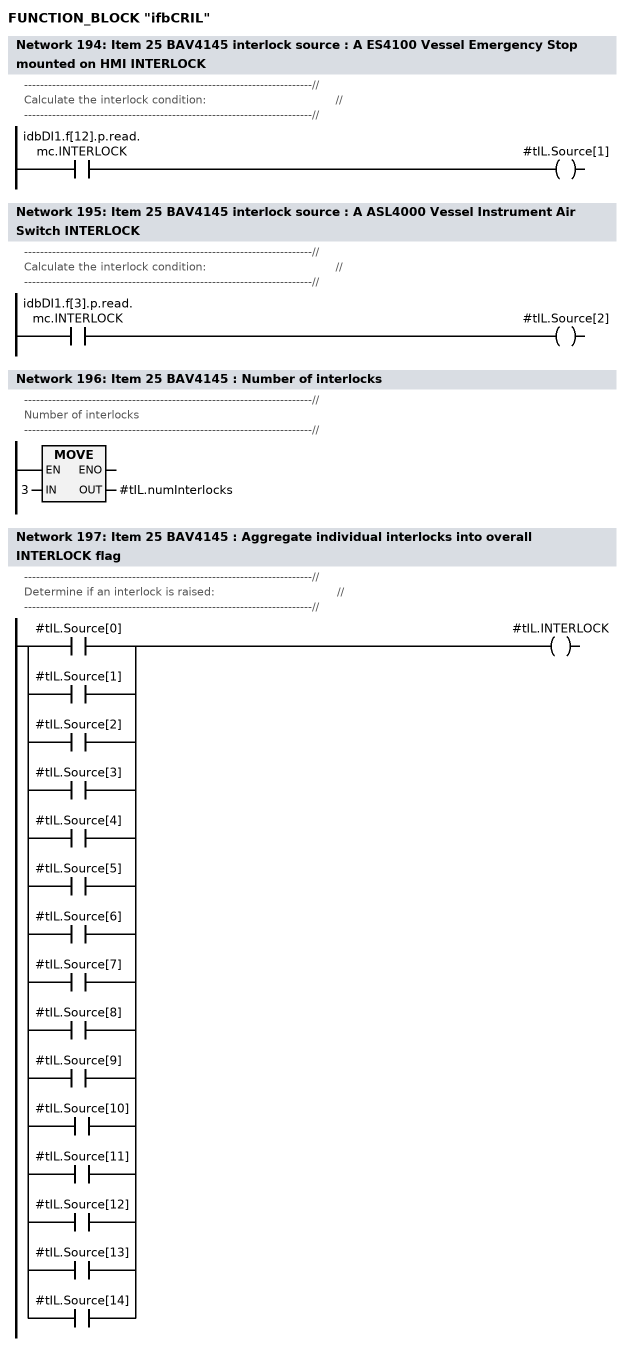
    A idbDI1.f[12].p.read.mc.INTERLOCK;
    = #tIL.Source[1];

NETWORK
TITLE = Item 25 BAV4145 interlock source : A ASL4000 Vessel Instrument Air Switch INTERLOCK
    //------------------------------------------------------------------------//
    // Calculate the interlock condition:                                     //
    //------------------------------------------------------------------------//
    A idbDI1.f[3].p.read.mc.INTERLOCK;
    = #tIL.Source[2];


NETWORK
TITLE = Item 25 BAV4145 : Number of interlocks
    //------------------------------------------------------------------------//
    // Number of interlocks
    //------------------------------------------------------------------------//
    L 3;
    T #tIL.numInterlocks;

NETWORK
TITLE = Item 25 BAV4145 : Aggregate individual interlocks into overall INTERLOCK flag
    //------------------------------------------------------------------------//
    // Determine if an interlock is raised:                                   //
    //------------------------------------------------------------------------//
    O #tIL.Source[0];
    O #tIL.Source[1];
    O #tIL.Source[2];
    O #tIL.Source[3];
    O #tIL.Source[4];
    O #tIL.Source[5];
    O #tIL.Source[6];
    O #tIL.Source[7];
    O #tIL.Source[8];
    O #tIL.Source[9];
    O #tIL.Source[10];
    O #tIL.Source[11];
    O #tIL.Source[12];
    O #tIL.Source[13];
    O #tIL.Source[14];
    = #tIL.INTERLOCK;

NETWORK
TITLE = Item 25 BAV4145 : Update the instance data
    //------------------------------------------------------------------------//
    // Update the instance DB with the calculated interlock flags:            //
    //------------------------------------------------------------------------//
    CALL MOVE
    {value_type := 'Variant'}
    (   IN                   := #tIL ,
        OUT                  := #p[25]
    );

NETWORK
TITLE = Item 26 BV1151 : MMFLx Cooling Water Supply Valve initialise variables
    //------------------------------------------------------------------------//
    // CRITICAL INTERLOCK   CRITICAL INTERLOCK   CRITICAL INTERLOCK   CRITICA //
    // CRITICAL INTERLOCK   CRITICAL INTERLOCK   CRITICAL INTERLOCK   CRITICA //
    //                                                                        //
    // Clear the interlock flag:                                              //
    //------------------------------------------------------------------------//
    A "alwaysLow";
    = #tIL.INTERLOCK;

    //------------------------------------------------------------------------//
    // Clear all interlock values to initialise them to off:                  //
    //------------------------------------------------------------------------//
    CALL FILL_BLK
    {value_type := 'Bool', count_type := 'UInt'}
    (   IN                   := 0 ,
        COUNT                := 15 ,
        OUT                  := #tIL.Source[0]
    );


NETWORK
TITLE = Item 26 BV1151 interlock source : AN BAV1167 Manufacturing Filtration Line Cooling Water Supply Drain Valve CLOSED   AN BAV1169 Manufacturing Filtration Line Cooling Water Return Drain Valve CLOSED
    //------------------------------------------------------------------------//
    // Calculate the interlock condition:                                     //
    //------------------------------------------------------------------------//
    AN(;
    L "idbPOS4".f[6].p.read.mc.STATE;
    L "dbCONST".BLK.POS4.STATE.CLOSED;
    ==I;
    );
AN(;
    L "idbPOS4".f[7].p.read.mc.STATE;
    L "dbCONST".BLK.POS4.STATE.CLOSED;
    ==I;
    );
    = #tIL.Source[0];

NETWORK
TITLE = Item 26 BV1151 interlock source : A RD1101 Vessel Burst Disc ALARM
    //------------------------------------------------------------------------//
    // Calculate the interlock condition:                                     //
    //------------------------------------------------------------------------//
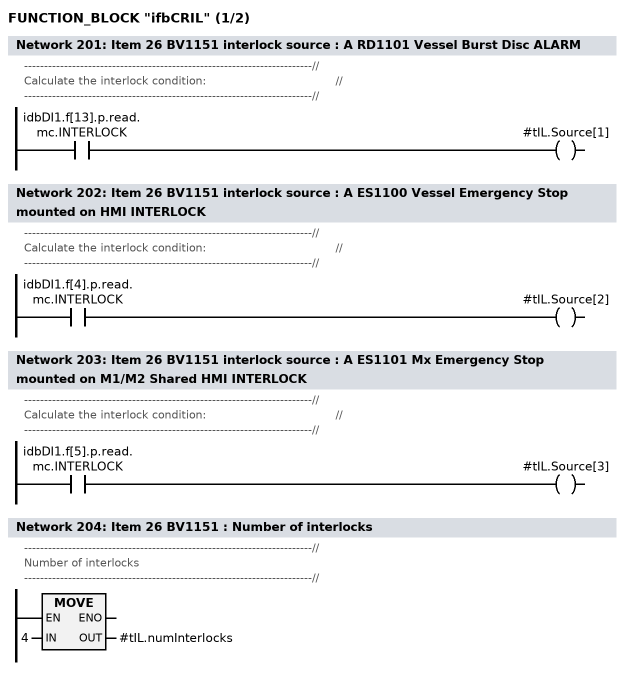
    A idbDI1.f[13].p.read.mc.INTERLOCK;
    = #tIL.Source[1];

NETWORK
TITLE = Item 26 BV1151 interlock source : A ES1100 Vessel Emergency Stop mounted on HMI INTERLOCK
    //------------------------------------------------------------------------//
    // Calculate the interlock condition:                                     //
    //------------------------------------------------------------------------//
    A idbDI1.f[4].p.read.mc.INTERLOCK;
    = #tIL.Source[2];

NETWORK
TITLE = Item 26 BV1151 interlock source : A ES1101 Mx Emergency Stop mounted on M1/M2 Shared HMI INTERLOCK
    //------------------------------------------------------------------------//
    // Calculate the interlock condition:                                     //
    //------------------------------------------------------------------------//
    A idbDI1.f[5].p.read.mc.INTERLOCK;
    = #tIL.Source[3];


NETWORK
TITLE = Item 26 BV1151 : Number of interlocks
    //------------------------------------------------------------------------//
    // Number of interlocks
    //------------------------------------------------------------------------//
    L 4;
    T #tIL.numInterlocks;

NETWORK
TITLE = Item 26 BV1151 : Aggregate individual interlocks into overall INTERLOCK flag
    //------------------------------------------------------------------------//
    // Determine if an interlock is raised:                                   //
    //------------------------------------------------------------------------//
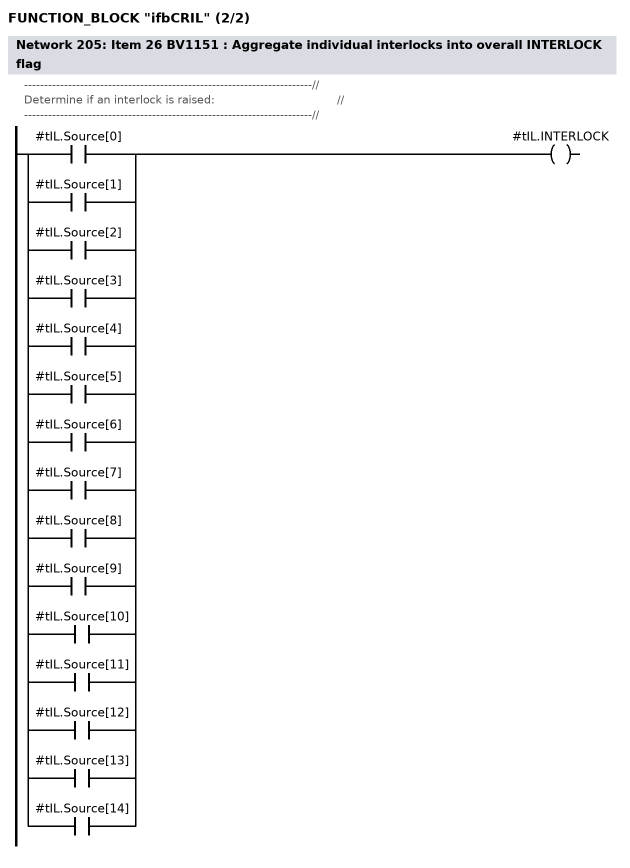
    O #tIL.Source[0];
    O #tIL.Source[1];
    O #tIL.Source[2];
    O #tIL.Source[3];
    O #tIL.Source[4];
    O #tIL.Source[5];
    O #tIL.Source[6];
    O #tIL.Source[7];
    O #tIL.Source[8];
    O #tIL.Source[9];
    O #tIL.Source[10];
    O #tIL.Source[11];
    O #tIL.Source[12];
    O #tIL.Source[13];
    O #tIL.Source[14];
    = #tIL.INTERLOCK;

NETWORK
TITLE = Item 26 BV1151 : Update the instance data
    //------------------------------------------------------------------------//
    // Update the instance DB with the calculated interlock flags:            //
    //------------------------------------------------------------------------//
    CALL MOVE
    {value_type := 'Variant'}
    (   IN                   := #tIL ,
        OUT                  := #p[26]
    );

NETWORK
TITLE = Item 27 BV1153 : MMFLx Cooling Water Return Valve initialise variables
    //------------------------------------------------------------------------//
    // CRITICAL INTERLOCK   CRITICAL INTERLOCK   CRITICAL INTERLOCK   CRITICA //
    // CRITICAL INTERLOCK   CRITICAL INTERLOCK   CRITICAL INTERLOCK   CRITICA //
    //                                                                        //
    // Clear the interlock flag:                                              //
    //------------------------------------------------------------------------//
    A "alwaysLow";
    = #tIL.INTERLOCK;

    //------------------------------------------------------------------------//
    // Clear all interlock values to initialise them to off:                  //
    //------------------------------------------------------------------------//
    CALL FILL_BLK
    {value_type := 'Bool', count_type := 'UInt'}
    (   IN                   := 0 ,
        COUNT                := 15 ,
        OUT                  := #tIL.Source[0]
    );


NETWORK
TITLE = Item 27 BV1153 interlock source : AN BAV1167 Manufacturing Filtration Line Cooling Water Supply Drain Valve CLOSED   AN BAV1169 Manufacturing Filtration Line Cooling Water Return Drain Valve CLOSED
    //------------------------------------------------------------------------//
    // Calculate the interlock condition:                                     //
    //------------------------------------------------------------------------//
    AN(;
    L "idbPOS4".f[6].p.read.mc.STATE;
    L "dbCONST".BLK.POS4.STATE.CLOSED;
    ==I;
    );
AN(;
    L "idbPOS4".f[7].p.read.mc.STATE;
    L "dbCONST".BLK.POS4.STATE.CLOSED;
    ==I;
    );
    = #tIL.Source[0];

NETWORK
TITLE = Item 27 BV1153 interlock source : A RD1101 Vessel Burst Disc ALARM
    //------------------------------------------------------------------------//
    // Calculate the interlock condition:                                     //
    //------------------------------------------------------------------------//
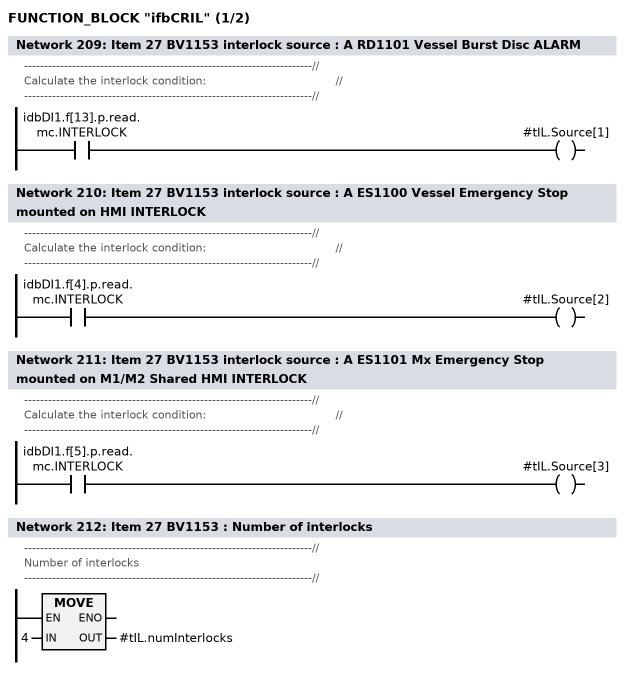
    A idbDI1.f[13].p.read.mc.INTERLOCK;
    = #tIL.Source[1];

NETWORK
TITLE = Item 27 BV1153 interlock source : A ES1100 Vessel Emergency Stop mounted on HMI INTERLOCK
    //------------------------------------------------------------------------//
    // Calculate the interlock condition:                                     //
    //------------------------------------------------------------------------//
    A idbDI1.f[4].p.read.mc.INTERLOCK;
    = #tIL.Source[2];

NETWORK
TITLE = Item 27 BV1153 interlock source : A ES1101 Mx Emergency Stop mounted on M1/M2 Shared HMI INTERLOCK
    //------------------------------------------------------------------------//
    // Calculate the interlock condition:                                     //
    //------------------------------------------------------------------------//
    A idbDI1.f[5].p.read.mc.INTERLOCK;
    = #tIL.Source[3];


NETWORK
TITLE = Item 27 BV1153 : Number of interlocks
    //------------------------------------------------------------------------//
    // Number of interlocks
    //------------------------------------------------------------------------//
    L 4;
    T #tIL.numInterlocks;

NETWORK
TITLE = Item 27 BV1153 : Aggregate individual interlocks into overall INTERLOCK flag
    //------------------------------------------------------------------------//
    // Determine if an interlock is raised:                                   //
    //------------------------------------------------------------------------//
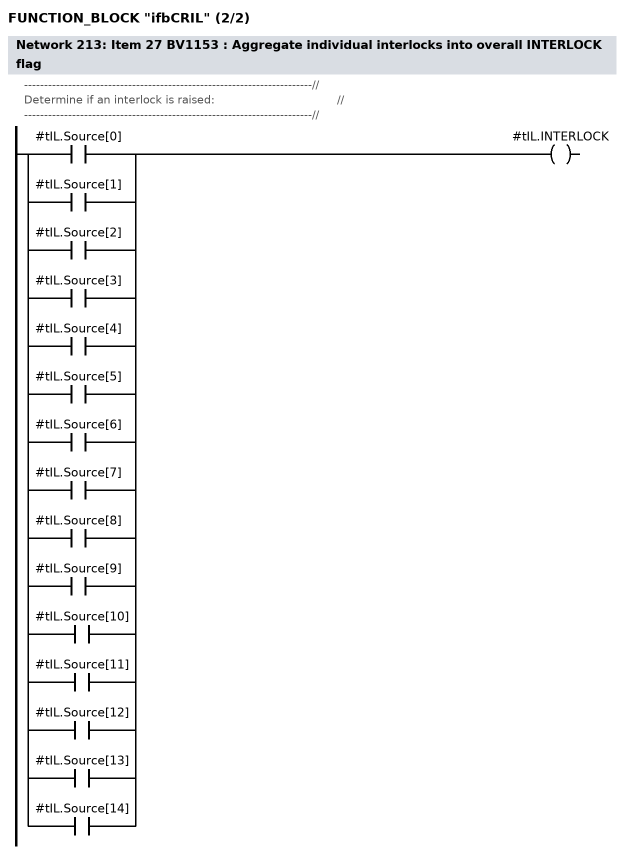
    O #tIL.Source[0];
    O #tIL.Source[1];
    O #tIL.Source[2];
    O #tIL.Source[3];
    O #tIL.Source[4];
    O #tIL.Source[5];
    O #tIL.Source[6];
    O #tIL.Source[7];
    O #tIL.Source[8];
    O #tIL.Source[9];
    O #tIL.Source[10];
    O #tIL.Source[11];
    O #tIL.Source[12];
    O #tIL.Source[13];
    O #tIL.Source[14];
    = #tIL.INTERLOCK;

NETWORK
TITLE = Item 27 BV1153 : Update the instance data
    //------------------------------------------------------------------------//
    // Update the instance DB with the calculated interlock flags:            //
    //------------------------------------------------------------------------//
    CALL MOVE
    {value_type := 'Variant'}
    (   IN                   := #tIL ,
        OUT                  := #p[27]
    );

NETWORK
TITLE = Item 28 BV2151 : MMFLx Cooling Water Supply Valve initialise variables
    //------------------------------------------------------------------------//
    // CRITICAL INTERLOCK   CRITICAL INTERLOCK   CRITICAL INTERLOCK   CRITICA //
    // CRITICAL INTERLOCK   CRITICAL INTERLOCK   CRITICAL INTERLOCK   CRITICA //
    //                                                                        //
    // Clear the interlock flag:                                              //
    //------------------------------------------------------------------------//
    A "alwaysLow";
    = #tIL.INTERLOCK;

    //------------------------------------------------------------------------//
    // Clear all interlock values to initialise them to off:                  //
    //------------------------------------------------------------------------//
    CALL FILL_BLK
    {value_type := 'Bool', count_type := 'UInt'}
    (   IN                   := 0 ,
        COUNT                := 15 ,
        OUT                  := #tIL.Source[0]
    );


NETWORK
TITLE = Item 28 BV2151 interlock source : AN BAV2167 Manufacturing Filtration Line Cooling Water Supply Drain Valve CLOSED   AN BAV2169 Manufacturing Filtration Line Cooling Water Return Drain Valve CLOSED
    //------------------------------------------------------------------------//
    // Calculate the interlock condition:                                     //
    //------------------------------------------------------------------------//
    AN(;
    L "idbPOS4".f[14].p.read.mc.STATE;
    L "dbCONST".BLK.POS4.STATE.CLOSED;
    ==I;
    );
AN(;
    L "idbPOS4".f[15].p.read.mc.STATE;
    L "dbCONST".BLK.POS4.STATE.CLOSED;
    ==I;
    );
    = #tIL.Source[0];

NETWORK
TITLE = Item 28 BV2151 interlock source : A RD2101 Vessel Burst Disc ALARM
    //------------------------------------------------------------------------//
    // Calculate the interlock condition:                                     //
    //------------------------------------------------------------------------//
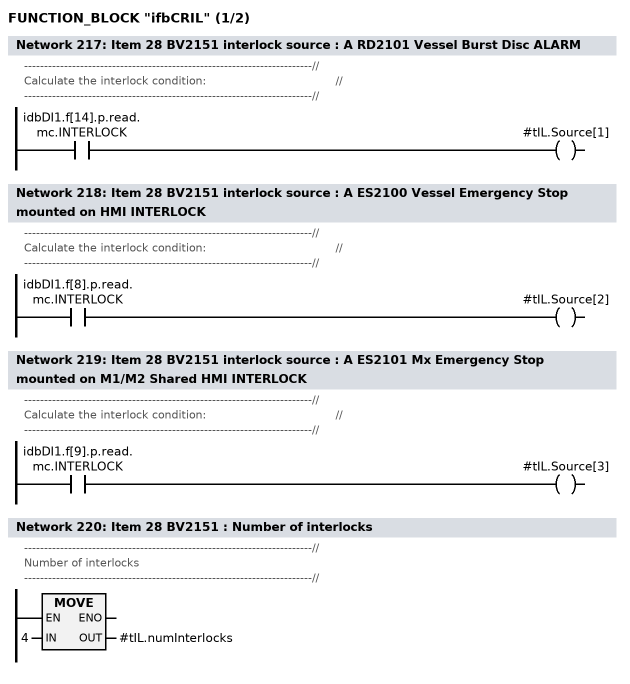
    A idbDI1.f[14].p.read.mc.INTERLOCK;
    = #tIL.Source[1];

NETWORK
TITLE = Item 28 BV2151 interlock source : A ES2100 Vessel Emergency Stop mounted on HMI INTERLOCK
    //------------------------------------------------------------------------//
    // Calculate the interlock condition:                                     //
    //------------------------------------------------------------------------//
    A idbDI1.f[8].p.read.mc.INTERLOCK;
    = #tIL.Source[2];

NETWORK
TITLE = Item 28 BV2151 interlock source : A ES2101 Mx Emergency Stop mounted on M1/M2 Shared HMI INTERLOCK
    //------------------------------------------------------------------------//
    // Calculate the interlock condition:                                     //
    //------------------------------------------------------------------------//
    A idbDI1.f[9].p.read.mc.INTERLOCK;
    = #tIL.Source[3];


NETWORK
TITLE = Item 28 BV2151 : Number of interlocks
    //------------------------------------------------------------------------//
    // Number of interlocks
    //------------------------------------------------------------------------//
    L 4;
    T #tIL.numInterlocks;

NETWORK
TITLE = Item 28 BV2151 : Aggregate individual interlocks into overall INTERLOCK flag
    //------------------------------------------------------------------------//
    // Determine if an interlock is raised:                                   //
    //------------------------------------------------------------------------//
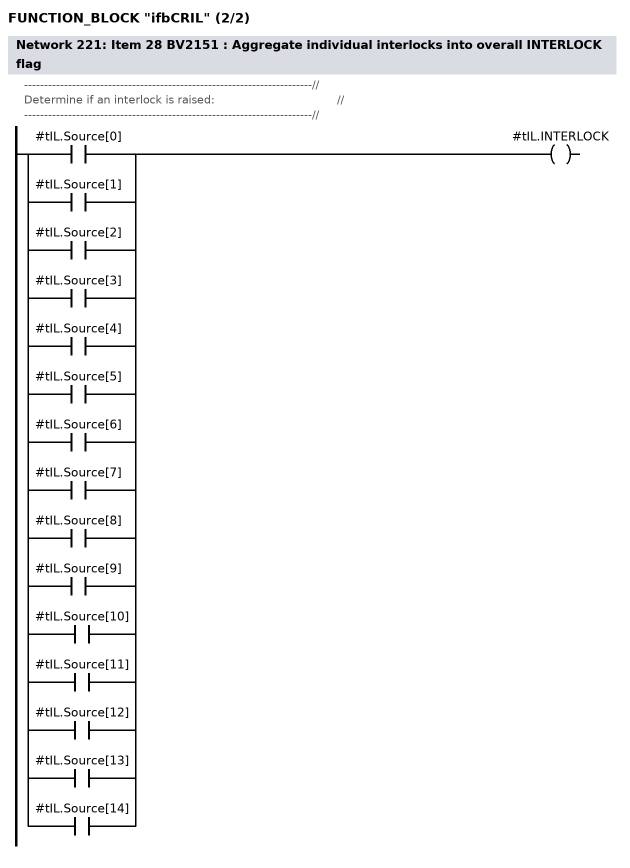
    O #tIL.Source[0];
    O #tIL.Source[1];
    O #tIL.Source[2];
    O #tIL.Source[3];
    O #tIL.Source[4];
    O #tIL.Source[5];
    O #tIL.Source[6];
    O #tIL.Source[7];
    O #tIL.Source[8];
    O #tIL.Source[9];
    O #tIL.Source[10];
    O #tIL.Source[11];
    O #tIL.Source[12];
    O #tIL.Source[13];
    O #tIL.Source[14];
    = #tIL.INTERLOCK;

NETWORK
TITLE = Item 28 BV2151 : Update the instance data
    //------------------------------------------------------------------------//
    // Update the instance DB with the calculated interlock flags:            //
    //------------------------------------------------------------------------//
    CALL MOVE
    {value_type := 'Variant'}
    (   IN                   := #tIL ,
        OUT                  := #p[28]
    );

NETWORK
TITLE = Item 29 BV2153 : MMFLx Cooling Water Return Valve initialise variables
    //------------------------------------------------------------------------//
    // CRITICAL INTERLOCK   CRITICAL INTERLOCK   CRITICAL INTERLOCK   CRITICA //
    // CRITICAL INTERLOCK   CRITICAL INTERLOCK   CRITICAL INTERLOCK   CRITICA //
    //                                                                        //
    // Clear the interlock flag:                                              //
    //------------------------------------------------------------------------//
    A "alwaysLow";
    = #tIL.INTERLOCK;

    //------------------------------------------------------------------------//
    // Clear all interlock values to initialise them to off:                  //
    //------------------------------------------------------------------------//
    CALL FILL_BLK
    {value_type := 'Bool', count_type := 'UInt'}
    (   IN                   := 0 ,
        COUNT                := 15 ,
        OUT                  := #tIL.Source[0]
    );


NETWORK
TITLE = Item 29 BV2153 interlock source : AN BAV2167 Manufacturing Filtration Line Cooling Water Supply Drain Valve CLOSED   AN BAV2169 Manufacturing Filtration Line Cooling Water Return Drain Valve CLOSED
    //------------------------------------------------------------------------//
    // Calculate the interlock condition:                                     //
    //------------------------------------------------------------------------//
    AN(;
    L "idbPOS4".f[14].p.read.mc.STATE;
    L "dbCONST".BLK.POS4.STATE.CLOSED;
    ==I;
    );
AN(;
    L "idbPOS4".f[15].p.read.mc.STATE;
    L "dbCONST".BLK.POS4.STATE.CLOSED;
    ==I;
    );
    = #tIL.Source[0];

NETWORK
TITLE = Item 29 BV2153 interlock source : A RD2101 Vessel Burst Disc ALARM
    //------------------------------------------------------------------------//
    // Calculate the interlock condition:                                     //
    //------------------------------------------------------------------------//
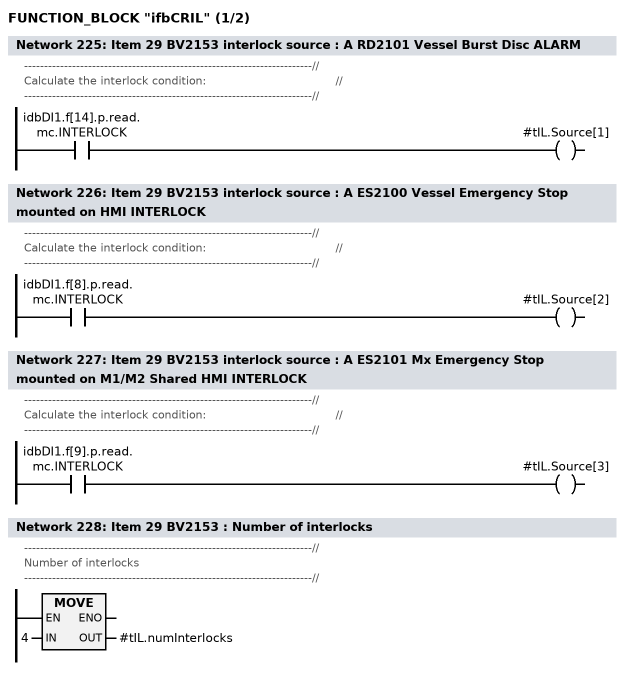
    A idbDI1.f[14].p.read.mc.INTERLOCK;
    = #tIL.Source[1];

NETWORK
TITLE = Item 29 BV2153 interlock source : A ES2100 Vessel Emergency Stop mounted on HMI INTERLOCK
    //------------------------------------------------------------------------//
    // Calculate the interlock condition:                                     //
    //------------------------------------------------------------------------//
    A idbDI1.f[8].p.read.mc.INTERLOCK;
    = #tIL.Source[2];

NETWORK
TITLE = Item 29 BV2153 interlock source : A ES2101 Mx Emergency Stop mounted on M1/M2 Shared HMI INTERLOCK
    //------------------------------------------------------------------------//
    // Calculate the interlock condition:                                     //
    //------------------------------------------------------------------------//
    A idbDI1.f[9].p.read.mc.INTERLOCK;
    = #tIL.Source[3];


NETWORK
TITLE = Item 29 BV2153 : Number of interlocks
    //------------------------------------------------------------------------//
    // Number of interlocks
    //------------------------------------------------------------------------//
    L 4;
    T #tIL.numInterlocks;

NETWORK
TITLE = Item 29 BV2153 : Aggregate individual interlocks into overall INTERLOCK flag
    //------------------------------------------------------------------------//
    // Determine if an interlock is raised:                                   //
    //------------------------------------------------------------------------//
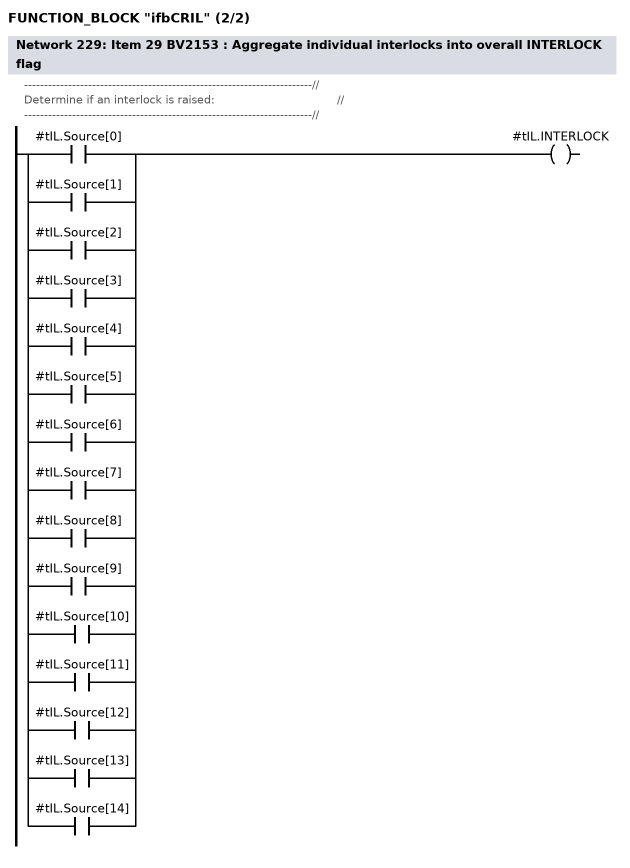
    O #tIL.Source[0];
    O #tIL.Source[1];
    O #tIL.Source[2];
    O #tIL.Source[3];
    O #tIL.Source[4];
    O #tIL.Source[5];
    O #tIL.Source[6];
    O #tIL.Source[7];
    O #tIL.Source[8];
    O #tIL.Source[9];
    O #tIL.Source[10];
    O #tIL.Source[11];
    O #tIL.Source[12];
    O #tIL.Source[13];
    O #tIL.Source[14];
    = #tIL.INTERLOCK;

NETWORK
TITLE = Item 29 BV2153 : Update the instance data
    //------------------------------------------------------------------------//
    // Update the instance DB with the calculated interlock flags:            //
    //------------------------------------------------------------------------//
    CALL MOVE
    {value_type := 'Variant'}
    (   IN                   := #tIL ,
        OUT                  := #p[29]
    );

NETWORK
TITLE = Item 30 DV1101 : Vent Valve initialise variables
    //------------------------------------------------------------------------//
    // CRITICAL INTERLOCK   CRITICAL INTERLOCK   CRITICAL INTERLOCK   CRITICA //
    // CRITICAL INTERLOCK   CRITICAL INTERLOCK   CRITICAL INTERLOCK   CRITICA //
    //                                                                        //
    // Clear the interlock flag:                                              //
    //------------------------------------------------------------------------//
    A "alwaysLow";
    = #tIL.INTERLOCK;

    //------------------------------------------------------------------------//
    // Clear all interlock values to initialise them to off:                  //
    //------------------------------------------------------------------------//
    CALL FILL_BLK
    {value_type := 'Bool', count_type := 'UInt'}
    (   IN                   := 0 ,
        COUNT                := 15 ,
        OUT                  := #tIL.Source[0]
    );


NETWORK
TITLE = Item 30 DV1101 interlock source : A RD1101 Vessel Burst Disc ALARM
    //------------------------------------------------------------------------//
    // Calculate the interlock condition:                                     //
    //------------------------------------------------------------------------//
    A idbDI1.f[13].p.read.mc.INTERLOCK;
    = #tIL.Source[0];

NETWORK
TITLE = Item 30 DV1101 interlock source : A ES1100 Vessel Emergency Stop mounted on HMI INTERLOCK
    //------------------------------------------------------------------------//
    // Calculate the interlock condition:                                     //
    //------------------------------------------------------------------------//
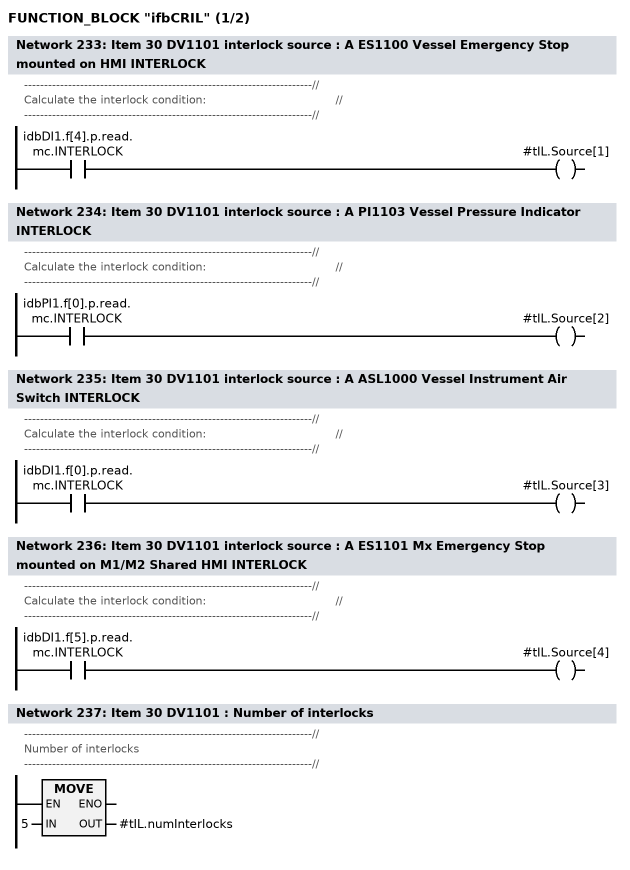
    A idbDI1.f[4].p.read.mc.INTERLOCK;
    = #tIL.Source[1];

NETWORK
TITLE = Item 30 DV1101 interlock source : A PI1103 Vessel Pressure Indicator INTERLOCK
    //------------------------------------------------------------------------//
    // Calculate the interlock condition:                                     //
    //------------------------------------------------------------------------//
    A idbPI1.f[0].p.read.mc.INTERLOCK;
    = #tIL.Source[2];

NETWORK
TITLE = Item 30 DV1101 interlock source : A ASL1000 Vessel Instrument Air Switch INTERLOCK
    //------------------------------------------------------------------------//
    // Calculate the interlock condition:                                     //
    //------------------------------------------------------------------------//
    A idbDI1.f[0].p.read.mc.INTERLOCK;
    = #tIL.Source[3];

NETWORK
TITLE = Item 30 DV1101 interlock source : A ES1101 Mx Emergency Stop mounted on M1/M2 Shared HMI INTERLOCK
    //------------------------------------------------------------------------//
    // Calculate the interlock condition:                                     //
    //------------------------------------------------------------------------//
    A idbDI1.f[5].p.read.mc.INTERLOCK;
    = #tIL.Source[4];


NETWORK
TITLE = Item 30 DV1101 : Number of interlocks
    //------------------------------------------------------------------------//
    // Number of interlocks
    //------------------------------------------------------------------------//
    L 5;
    T #tIL.numInterlocks;

NETWORK
TITLE = Item 30 DV1101 : Aggregate individual interlocks into overall INTERLOCK flag
    //------------------------------------------------------------------------//
    // Determine if an interlock is raised:                                   //
    //------------------------------------------------------------------------//
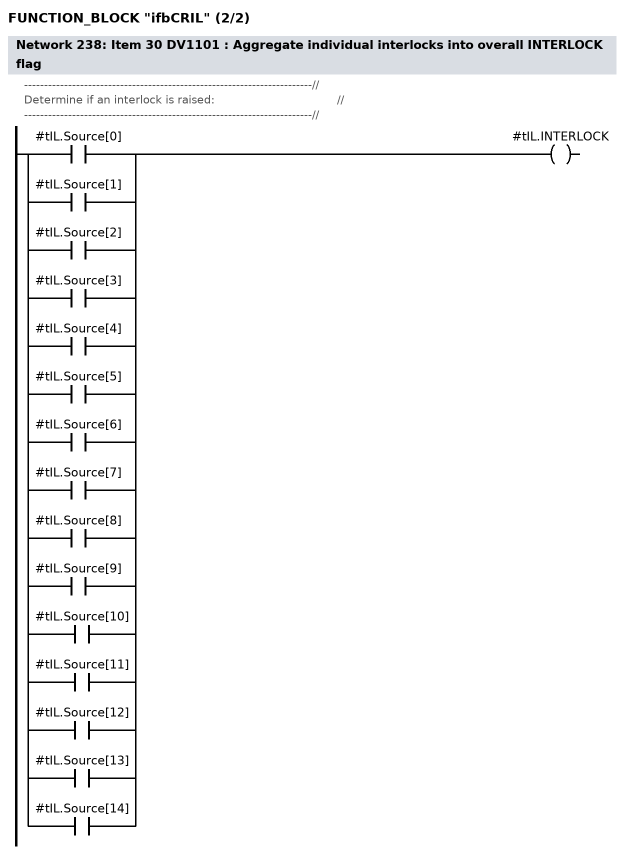
    O #tIL.Source[0];
    O #tIL.Source[1];
    O #tIL.Source[2];
    O #tIL.Source[3];
    O #tIL.Source[4];
    O #tIL.Source[5];
    O #tIL.Source[6];
    O #tIL.Source[7];
    O #tIL.Source[8];
    O #tIL.Source[9];
    O #tIL.Source[10];
    O #tIL.Source[11];
    O #tIL.Source[12];
    O #tIL.Source[13];
    O #tIL.Source[14];
    = #tIL.INTERLOCK;

NETWORK
TITLE = Item 30 DV1101 : Update the instance data
    //------------------------------------------------------------------------//
    // Update the instance DB with the calculated interlock flags:            //
    //------------------------------------------------------------------------//
    CALL MOVE
    {value_type := 'Variant'}
    (   IN                   := #tIL ,
        OUT                  := #p[30]
    );

NETWORK
TITLE = Item 31 DV1103 : HP CA Supply Valve initialise variables
    //------------------------------------------------------------------------//
    // CRITICAL INTERLOCK   CRITICAL INTERLOCK   CRITICAL INTERLOCK   CRITICA //
    // CRITICAL INTERLOCK   CRITICAL INTERLOCK   CRITICAL INTERLOCK   CRITICA //
    //                                                                        //
    // Clear the interlock flag:                                              //
    //------------------------------------------------------------------------//
    A "alwaysLow";
    = #tIL.INTERLOCK;

    //------------------------------------------------------------------------//
    // Clear all interlock values to initialise them to off:                  //
    //------------------------------------------------------------------------//
    CALL FILL_BLK
    {value_type := 'Bool', count_type := 'UInt'}
    (   IN                   := 0 ,
        COUNT                := 15 ,
        OUT                  := #tIL.Source[0]
    );


NETWORK
TITLE = Item 31 DV1103 interlock source : A RD1101 Vessel Burst Disc ALARM
    //------------------------------------------------------------------------//
    // Calculate the interlock condition:                                     //
    //------------------------------------------------------------------------//
    A idbDI1.f[13].p.read.mc.INTERLOCK;
    = #tIL.Source[0];

NETWORK
TITLE = Item 31 DV1103 interlock source : A ES1100 Vessel Emergency Stop mounted on HMI INTERLOCK
    //------------------------------------------------------------------------//
    // Calculate the interlock condition:                                     //
    //------------------------------------------------------------------------//
